DATA_BLOCK "Timer"   // DB2
{ S7_Optimized_Access := 'TRUE' }
VERSION : 0.0
// stored: AutoNumber false, IsOnlyStoredInLoadMemory false, IsRetainMemResEnabled false, IsWriteProtectedInAS false, MemoryReserve 100
   VAR
      T0 { S7_SetPoint := 'True'} : IEC_TIMER;   // Delay on pallet positioning
      T1 { S7_SetPoint := 'True'} : IEC_TIMER;   // Timer for acoustic siren
      T2 { S7_SetPoint := 'True'} : IEC_TIMER;   // Timer for restart after emergency
      T3 { S7_SetPoint := 'True'} : IEC_TIMER;   // Timer to reset emergency
      T4 { S7_SetPoint := 'True'} : IEC_TIMER;   // Timer to reset the cycles
      T5 { S7_SetPoint := 'True'} : IEC_TIMER;   // Delay for backward on table rotation inverter
      T6 { S7_SetPoint := 'True'} : IEC_TIMER;   // Delay for forward on table rotation inverter
      T7 { S7_SetPoint := 'True'} : IEC_TIMER;   // Timeout for table phase
      T8 { S7_SetPoint := 'True'} : IEC_TIMER;   // Table rotation speed timer
      T9 { S7_SetPoint := 'True'} : IEC_TIMER;   // Timer SA type for spool carriage motor
      T10 { S7_SetPoint := 'True'} : IEC_TIMER;   // Timer SA type for table rotation motor
      T11 { S7_SetPoint := 'True'} : IEC_TIMER;   // Timer SA type for spool carriage downward
      T12 { S7_SetPoint := 'True'} : IEC_TIMER;   // Timer SA type for spool carriage upward
      T13 { S7_SetPoint := 'True'} : IEC_TIMER;   // Timer SA type for top carriage motor
      T14 { S7_SetPoint := 'True'} : IEC_TIMER;   // Delay for forward on spool carriage and machine conveyor inverter
      T15 { S7_SetPoint := 'True'} : IEC_TIMER;   // Timer for lifter upward
      T16 { S7_SetPoint := 'True'} : IEC_TIMER;   // Timeout for pallet lifter upward/downward
      T17 { S7_SetPoint := 'True'} : IEC_TIMER;   // Time for pressure plate downward
      T18 { S7_SetPoint := 'True'} : IEC_TIMER;   // Timeout for pressure plate upward/downward
      T19 { S7_SetPoint := 'True'} : IEC_TIMER;   // Delay for backward on spool carriage and machine conveyor inverter
      T20 { S7_SetPoint := 'True'} : IEC_TIMER;   // Delay for table rotation deceleration
      T21 { S7_SetPoint := 'True'} : IEC_TIMER;   // Film broken delay for spool carriage
      T22 { S7_SetPoint := 'True'} : IEC_TIMER;   // Delay for pressure plate positioning on pallet
      T23 { S7_SetPoint := 'True'} : IEC_TIMER;   // Timer SA type for conveyor motor
      T24 { S7_SetPoint := 'True'} : IEC_TIMER;   // Delay on pallet positioning left
      T25 { S7_SetPoint := 'True'} : IEC_TIMER;   // Delay on machine conveyor stop
      T26 { S7_SetPoint := 'True'} : IEC_TIMER;   // Delay to load/unload pallet simultaneously
      T27 { S7_SetPoint := 'True'} : IEC_TIMER;   // Delay to have outfeed control free
      T28 { S7_SetPoint := 'True'} : IEC_TIMER;   // Timer for end of transfer signal
      T29 { S7_SetPoint := 'True'} : IEC_TIMER;   // Timer to check spool carriage encoder
      T30 { S7_SetPoint := 'True'} : IEC_TIMER;   // Timer to check spool carriage encoder
      T31 { S7_SetPoint := 'True'} : IEC_TIMER;   // Time to record spool carriage movement speed
      T32 { S7_SetPoint := 'True'} : IEC_TIMER;   // Timeout for single or lower(double) rope unit open/close
      T33 { S7_SetPoint := 'True'} : IEC_TIMER;   // Timer for outfeed rotating table control engaged
      T34 { S7_SetPoint := 'True'} : IEC_TIMER;   // Timer for prestretch restart
      T35 { S7_SetPoint := 'True'} : IEC_TIMER;   // Delay to open single or lower(double) rope unit
      T36 { S7_SetPoint := 'True'} : IEC_TIMER;   // Timeout for welder unit upward/downward
      T37 { S7_SetPoint := 'True'} : IEC_TIMER;   // Timeout for welder contrast downward
      T38 { S7_SetPoint := 'True'} : IEC_TIMER;   // Timeout for welder contrast upward
      T39 { S7_SetPoint := 'True'} : IEC_TIMER;   // Timeout for clamp upward/downward
      T40 { S7_SetPoint := 'True'} : IEC_TIMER;   // Timeout for clamp open/close
      T41 { S7_SetPoint := 'True'} : IEC_TIMER;   // Welding timer for welder
      T42 { S7_SetPoint := 'True'} : IEC_TIMER;   // Cutting timer
      T43 { S7_SetPoint := 'True'} : IEC_TIMER;   // Welder cooler timer
      T44 { S7_SetPoint := 'True'} : IEC_TIMER;   // Timer to check welder circuit 1 (current on)
      T45 { S7_SetPoint := 'True'} : IEC_TIMER;   // Timer to check welder circuit 2 (current off)
      T46 { S7_SetPoint := 'True'} : IEC_TIMER;   // Spring clamp up
      T47 { S7_SetPoint := 'True'} : IEC_TIMER;   // Welder contrast up
      T48 { S7_SetPoint := 'True'} : IEC_TIMER;   // Spring clamp open
      T49 { S7_SetPoint := 'True'} : IEC_TIMER;   // Welder and cut unit up
      T50 { S7_SetPoint := 'True'} : IEC_TIMER;   // Timer for encoder check
      T51 { S7_SetPoint := 'True'} : IEC_TIMER;   // Timer for display comunication control
      T52 { S7_SetPoint := 'True'} : IEC_TIMER;   // Timer to return to page 1 after 3 minutes
      T53 { S7_SetPoint := 'True'} : IEC_TIMER;   // Delay for test cycle
      T54 { S7_SetPoint := 'True'} : IEC_TIMER;   // Timer to reset infeed safety barrier
      T55 { S7_SetPoint := 'True'} : IEC_TIMER;   // Timer to reset infeed safety barrier
      T56 { S7_SetPoint := 'True'} : IEC_TIMER;   // Timer to reset outfeed safety barrier
      T57 { S7_SetPoint := 'True'} : IEC_TIMER;   // Timer to reset outfeed safety barrier
      T58 { S7_SetPoint := 'True'} : IEC_TIMER;   // Delay for infeed safety barrier muting photocell
      T59 { S7_SetPoint := 'True'} : IEC_TIMER;   // Delay for outfeed safety barrier muting photocell
      T60 { S7_SetPoint := 'True'} : IEC_TIMER;   // Delay for spool carriage downward for film tail
      T61 { S7_SetPoint := 'True'} : IEC_TIMER;   // Delay to open clamp during wrapping cycle
      T62 { S7_SetPoint := 'True'} : IEC_TIMER;   // Timer for table rotation forward on twist
      T63 { S7_SetPoint := 'True'} : IEC_TIMER;   // Timer SA type for top carriage upward
      T64 { S7_SetPoint := 'True'} : IEC_TIMER;   // Timer SA type for top carriage downward
      T65 { S7_SetPoint := 'True'} : IEC_TIMER;   // Delay on safety for top carriage movement
      T66 { S7_SetPoint := 'True'} : IEC_TIMER;   // Timer to check top film presence
      T67 { S7_SetPoint := 'True'} : IEC_TIMER;   // Timer to check top film presence
      T68 { S7_SetPoint := 'True'} : IEC_TIMER;   // Timeout for top film cutter forward/backward
      T69 { S7_SetPoint := 'True'} : IEC_TIMER;   // Timeout for clamp to lift top film open/close
      T70 { S7_SetPoint := 'True'} : IEC_TIMER;   // Timeout for clamp to block top film open/close
      T71 { S7_SetPoint := 'True'} : IEC_TIMER;   // Timeout for top carriage forward/backward movement
      T72 { S7_SetPoint := 'True'} : IEC_TIMER;   // Timeout for top carriage forward/backward movement
      T73 { S7_SetPoint := 'True'} : IEC_TIMER;   // Timeout for top carriage upward/downward movement
      T74 { S7_SetPoint := 'True'} : IEC_TIMER;   // Timeout for top carriage upward/downward movement
      T75 { S7_SetPoint := 'True'} : IEC_TIMER;   // Delay for spool carriage downward during top cycle
      T76 { S7_SetPoint := 'True'} : IEC_TIMER;   // Claw clamp closed
      T77 { S7_SetPoint := 'True'} : IEC_TIMER;   // Timeout for welder and cut unit forward/backward
      T78 { S7_SetPoint := 'True'} : IEC_TIMER;   // Delay to open upper(double) rope unit
      T79 { S7_SetPoint := 'True'} : IEC_TIMER;   // Timer SA type for table rotation brake
      T80 { S7_SetPoint := 'True'} : IEC_TIMER;   // Timer for spool carriage movement speed
      T81 { S7_SetPoint := 'True'} : IEC_TIMER;   // Claw clamp closed
      T82 { S7_SetPoint := 'True'} : IEC_TIMER;   // Timeout for welder and cut unit forward/backward
      T83 { S7_SetPoint := 'True'} : IEC_TIMER;   // Delay between airblow and clamp
      T84 { S7_SetPoint := 'True'} : IEC_TIMER;   // Timer for table rotation speed
      T85 { S7_SetPoint := 'True'} : IEC_TIMER;   // Delay on infeed conveyor stop
      T86 { S7_SetPoint := 'True'} : IEC_TIMER;   // Delay for prestretch during acceleration
      T87 { S7_SetPoint := 'True'} : IEC_TIMER;   // Timer for slow conveyor manual movement
      T88 { S7_SetPoint := 'True'} : IEC_TIMER;
      T89 { S7_SetPoint := 'True'} : IEC_TIMER;   // Timer for wrong pallet positioning without outfeed control
      T90 { S7_SetPoint := 'True'} : IEC_TIMER;   // Timer for spool carriage upward for table cycle
      T91 { S7_SetPoint := 'True'} : IEC_TIMER;   // Delay to close clamp after cutter forward
      T92 { S7_SetPoint := 'True'} : IEC_TIMER;   // Delay for contrast downward
      T93 { S7_SetPoint := 'True'} : IEC_TIMER;
      T94 { S7_SetPoint := 'True'} : IEC_TIMER;
      T95 { S7_SetPoint := 'True'} : IEC_TIMER;
      T96 { S7_SetPoint := 'True'} : IEC_TIMER;   // Timeout for fire door pos.4-5 opening
      T97 { S7_SetPoint := 'True'} : IEC_TIMER;   // Delay conveyor manual movement
      T98 { S7_SetPoint := 'True'} : IEC_TIMER;   // Delay start cycle pos.1
      T99 { S7_SetPoint := 'True'} : IEC_TIMER;   // Time to load with forklift
      T100 { S7_SetPoint := 'True'} : IEC_TIMER;   // Timer for end of pallet transfer in infeed signal
      T101 { S7_SetPoint := 'True'} : IEC_TIMER;   // Timeout for conveyor pos 01
      T102 { S7_SetPoint := 'True'} : IEC_TIMER;   // Time to load with forklift
      T103 { S7_SetPoint := 'True'} : IEC_TIMER;   // Timeout for conveyor pos 02
      T104 { S7_SetPoint := 'True'} : IEC_TIMER;
      T105 { S7_SetPoint := 'True'} : IEC_TIMER;   // Timeout for conveyor pos 04
      T106 { S7_SetPoint := 'True'} : IEC_TIMER;   // Timeout for conveyor pos 03
      T107 { S7_SetPoint := 'True'} : IEC_TIMER;   // Time for pallet unload with forklift
      T108 { S7_SetPoint := 'True'} : IEC_TIMER;   // Delay Button Stop cycle support memory
      T109 { S7_SetPoint := 'True'} : IEC_TIMER;   // Time for pallet load with forklift from reverse
      T110 { S7_SetPoint := 'True'} : IEC_TIMER;   // Timer to reset machine and cycle
      T111 { S7_SetPoint := 'True'} : IEC_TIMER;   // Delay timer for lifter pos.2 low position
      T112 { S7_SetPoint := 'True'} : IEC_TIMER;   // Delay timer for lifter pos.2 up position
      T113 { S7_SetPoint := 'True'} : IEC_TIMER;   // Delay timer pallet positioned on lifter pos.2
      T114 { S7_SetPoint := 'True'} : IEC_TIMER;   // Timer SA for lifter in top position
      T115 { S7_SetPoint := 'True'} : IEC_TIMER;   // Timeout for conveyor pos.2
      T116 { S7_SetPoint := 'True'} : IEC_TIMER;   // Timeout for lifter pos.2 upstroke
      T117 { S7_SetPoint := 'True'} : IEC_TIMER;   // Timeout for lifter pos.2 downstroke
      T118 { S7_SetPoint := 'True'} : IEC_TIMER;   // Timer to filter lifter pos.2 in up position
      T119 { S7_SetPoint := 'True'} : IEC_TIMER;
      T120 { S7_SetPoint := 'True'} : IEC_TIMER;   // Timer to check conveyor encoder
      T121 { S7_SetPoint := 'True'} : IEC_TIMER;   // Timer to check conveyor encoder
      T122 { S7_SetPoint := 'True'} : IEC_TIMER;
      T123 { S7_SetPoint := 'True'} : IEC_TIMER;
      T124 { S7_SetPoint := 'True'} : IEC_TIMER;
      T125 { S7_SetPoint := 'True'} : IEC_TIMER;
      T126 { S7_SetPoint := 'True'} : IEC_TIMER;
      T127 { S7_SetPoint := 'True'} : IEC_TIMER;   // Delay to have outfeed rotating arm control free from reverse
      T128 { S7_SetPoint := 'True'} : IEC_TIMER;   // Timer for end of transfer signal from reverse
      T129 { S7_SetPoint := 'True'} : IEC_TIMER;
      T130 { S7_SetPoint := 'True'} : IEC_TIMER;
      T131 { S7_SetPoint := 'True'} : IEC_TIMER;
      T132 { S7_SetPoint := 'True'} : IEC_TIMER;   // Timeout for single or lower(double) rope unit open/close
      T133 { S7_SetPoint := 'True'} : IEC_TIMER;
      T134 { S7_SetPoint := 'True'} : IEC_TIMER;
      T135 { S7_SetPoint := 'True'} : IEC_TIMER;   // Delay to open single or lower(double) rope unit
      T136 { S7_SetPoint := 'True'} : IEC_TIMER;
      T137 { S7_SetPoint := 'True'} : IEC_TIMER;
      T138 { S7_SetPoint := 'True'} : IEC_TIMER;
      T139 { S7_SetPoint := 'True'} : IEC_TIMER;   // Delay for top carriage forward stop (Top)
      T140 { S7_SetPoint := 'True'} : IEC_TIMER;   // Delay for top carriage backward stop (Top)
      T141 { S7_SetPoint := 'True'} : IEC_TIMER;
      T142 { S7_SetPoint := 'True'} : IEC_TIMER;   // Delay for top carriage down to release top film (Top)
      T143 { S7_SetPoint := 'True'} : IEC_TIMER;   // Delay to release top film from clamp (Top)
      T144 { S7_SetPoint := 'True'} : IEC_TIMER;   // Timer 1 for top film broken (Top)
      T145 { S7_SetPoint := 'True'} : IEC_TIMER;   // Timer 2 for top film broken (Top)
      T146 { S7_SetPoint := 'True'} : IEC_TIMER;   // Delay to stop top carriage forward for top film broken (Top)
      T147 { S7_SetPoint := 'True'} : IEC_TIMER;   // Delay to stop top carriage against vibration (Top)
      T148 { S7_SetPoint := 'True'} : IEC_TIMER;   // Timeout for top cutter (Top)
      T149 { S7_SetPoint := 'True'} : IEC_TIMER;   // Timeout for clamp to pull top film (Top)
      T150 { S7_SetPoint := 'True'} : IEC_TIMER;   // Timeout for clamp to block top film (Top)
      T151 { S7_SetPoint := 'True'} : IEC_TIMER;   // Timer SA type for top brake (Top)
      T152 { S7_SetPoint := 'True'} : IEC_TIMER;   // Timer for top brake control (Top)
      T153 { S7_SetPoint := 'True'} : IEC_TIMER;
      T154 { S7_SetPoint := 'True'} : IEC_TIMER;
      T155 { S7_SetPoint := 'True'} : IEC_TIMER;   // Timeout for conveyor pos 03
      T156 { S7_SetPoint := 'True'} : IEC_TIMER;   // Timeout for conveyor pos 04
      T157 { S7_SetPoint := 'True'} : IEC_TIMER;   // Timeout for conveyor pos 05
      T158 { S7_SetPoint := 'True'} : IEC_TIMER;   // Timeout for conveyor pos 06
      T159 { S7_SetPoint := 'True'} : IEC_TIMER;   // Timeout for conveyor pos 07
      T160 { S7_SetPoint := 'True'} : IEC_TIMER;   // Timeout for conveyor pos 08
      T161 { S7_SetPoint := 'True'} : IEC_TIMER;
      T162 { S7_SetPoint := 'True'} : IEC_TIMER;
      T163 { S7_SetPoint := 'True'} : IEC_TIMER;   // Watchdog timer for network communication
      T164 { S7_SetPoint := 'True'} : IEC_TIMER;
      T165 { S7_SetPoint := 'True'} : IEC_TIMER;
      T166 { S7_SetPoint := 'True'} : IEC_TIMER;
      T167 { S7_SetPoint := 'True'} : IEC_TIMER;
      T168 { S7_SetPoint := 'True'} : IEC_TIMER;
      T169 { S7_SetPoint := 'True'} : IEC_TIMER;
      T170 { S7_SetPoint := 'True'} : IEC_TIMER;
      T171 { S7_SetPoint := 'True'} : IEC_TIMER;
      T172 { S7_SetPoint := 'True'} : IEC_TIMER;
      T173 { S7_SetPoint := 'True'} : IEC_TIMER;
      T174 { S7_SetPoint := 'True'} : IEC_TIMER;
      T175 { S7_SetPoint := 'True'} : IEC_TIMER;
      T176 { S7_SetPoint := 'True'} : IEC_TIMER;
      T177 { S7_SetPoint := 'True'} : IEC_TIMER;
      T178 { S7_SetPoint := 'True'} : IEC_TIMER;
      T179 { S7_SetPoint := 'True'} : IEC_TIMER;   // Delay for top pallet height reading photocell (fast cycle)
      T180 { S7_SetPoint := 'True'} : IEC_TIMER;
      T181 { S7_SetPoint := 'True'} : IEC_TIMER;
      T182 { S7_SetPoint := 'True'} : IEC_TIMER;
      T183 { S7_SetPoint := 'True'} : IEC_TIMER;
      T184 { S7_SetPoint := 'True'} : IEC_TIMER;
      T185 { S7_SetPoint := 'True'} : IEC_TIMER;
      T186 { S7_SetPoint := 'True'} : IEC_TIMER;
      T187 { S7_SetPoint := 'True'} : IEC_TIMER;
      T188 { S7_SetPoint := 'True'} : IEC_TIMER;
      T189 { S7_SetPoint := 'True'} : IEC_TIMER;
      T190 { S7_SetPoint := 'True'} : IEC_TIMER;
      T191 { S7_SetPoint := 'True'} : IEC_TIMER;
      T192 { S7_SetPoint := 'True'} : IEC_TIMER;
      T193 { S7_SetPoint := 'True'} : IEC_TIMER;
      T194 { S7_SetPoint := 'True'} : IEC_TIMER;
      T195 { S7_SetPoint := 'True'} : IEC_TIMER;
      T196 { S7_SetPoint := 'True'} : IEC_TIMER;
      T197 { S7_SetPoint := 'True'} : IEC_TIMER;
      T198 { S7_SetPoint := 'True'} : IEC_TIMER;
      T199 { S7_SetPoint := 'True'} : IEC_TIMER;
      T200 { S7_SetPoint := 'True'} : IEC_TIMER;   // T_InverterAlarm - Time to filter inverter alarms
      T201 { S7_SetPoint := 'True'} : IEC_TIMER;   // T_ProfinetDiag - Time to filter 'DeviceStates' diagnostic output (Profinet)
      T202 { S7_SetPoint := 'True'} : IEC_TIMER;   // Timer for U201 start command (after enable)
      T203 { S7_SetPoint := 'True'} : IEC_TIMER;   // Timer table backward
      T204 { S7_SetPoint := 'True'} : IEC_TIMER;   // Timer ciclo fiera
      T205 { S7_SetPoint := 'True'} : IEC_TIMER;   // TON per OFF1 U201
      T206 { S7_SetPoint := 'True'} : IEC_TIMER;   // TOF per OFF1 U201
      T207 { S7_SetPoint := 'True'} : IEC_TIMER;   // Timer coppia tavola
      T208 { S7_SetPoint := 'True'} : IEC_TIMER;   // T_ModbusErrors
      T209 { S7_SetPoint := 'True'} : IEC_TIMER;
      T210 { S7_SetPoint := 'True'} : IEC_TIMER;   // Time to filter contrast back sensor
      T211 { S7_SetPoint := 'True'} : IEC_TIMER;   // Timeout for welder contrast forward
      T212 { S7_SetPoint := 'True'} : IEC_TIMER;   // Timeout for welder contrast backward
      T213 { S7_SetPoint := 'True'} : IEC_TIMER;   // Timeout for (double) full rope unit open/close
      T214 { S7_SetPoint := 'True'} : IEC_TIMER;   // Delay to open single or lower(double) rope unit
      T215 { S7_SetPoint := 'True'} : IEC_TIMER;   // Time Contrast Backward
      T216 { S7_SetPoint := 'True'} : IEC_TIMER;   // Time Contrast Manual forward
   END_VAR
BEGIN
   T0.PT := T#0MS;
   T0.IN := FALSE;
   T1.PT := T#1S_200MS;
   T1.IN := FALSE;
   T2.PT := T#6S;
   T2.IN := TRUE;
   T3.PT := T#700MS;
   T3.IN := FALSE;
   T4.PT := T#2S;
   T4.IN := FALSE;
   T5.PT := T#800MS;
   T5.IN := FALSE;
   T6.PT := T#800MS;
   T6.IN := FALSE;
   T7.PT := T#50S;
   T7.IN := FALSE;
   T8.PT := T#1M_39S;
   T8.IN := FALSE;
   T9.PT := T#700MS;
   T9.IN := FALSE;
   T10.PT := T#2S;
   T10.IN := FALSE;
   T11.PT := T#500MS;
   T11.IN := FALSE;
   T12.PT := T#500MS;
   T12.IN := FALSE;
   T13.PT := T#0MS;
   T13.IN := FALSE;
   T14.PT := T#200MS;
   T14.IN := FALSE;
   T15.PT := T#0MS;
   T15.IN := FALSE;
   T16.PT := T#0MS;
   T16.IN := FALSE;
   T17.PT := T#0MS;
   T17.IN := FALSE;
   T18.PT := T#0MS;
   T18.IN := FALSE;
   T19.PT := T#200MS;
   T19.IN := FALSE;
   T20.PT := T#0MS;
   T20.IN := FALSE;
   T21.PT := T#2S;
   T21.IN := FALSE;
   T22.PT := T#0MS;
   T22.IN := FALSE;
   T23.PT := T#0MS;
   T23.IN := FALSE;
   T24.PT := T#0MS;
   T24.IN := FALSE;
   T25.PT := T#0MS;
   T25.IN := FALSE;
   T26.PT := T#0MS;
   T26.IN := FALSE;
   T27.PT := T#1S_500MS;
   T27.IN := TRUE;
   T28.PT := T#2S;
   T28.IN := TRUE;
   T29.PT := T#0MS;
   T29.IN := FALSE;
   T30.PT := T#3S;
   T30.IN := FALSE;
   T31.PT := T#0MS;
   T31.IN := FALSE;
   T32.PT := T#0MS;
   T32.IN := FALSE;
   T33.PT := T#0MS;
   T33.IN := FALSE;
   T34.PT := T#0MS;
   T34.IN := FALSE;
   T35.PT := T#0MS;
   T35.IN := FALSE;
   T36.PT := T#0MS;
   T36.IN := FALSE;
   T37.PT := T#0MS;
   T37.IN := FALSE;
   T38.PT := T#10S;
   T38.IN := FALSE;
   T39.PT := T#0MS;
   T39.IN := FALSE;
   T40.PT := T#0MS;
   T40.IN := FALSE;
   T41.PT := T#650MS;
   T41.IN := FALSE;
   T42.PT := T#3S;
   T42.IN := FALSE;
   T43.PT := T#0MS;
   T43.IN := FALSE;
   T44.PT := T#3S_500MS;
   T44.IN := FALSE;
   T45.PT := T#1S;
   T45.IN := FALSE;
   T46.PT := T#0MS;
   T46.IN := FALSE;
   T47.PT := T#500MS;
   T47.IN := TRUE;
   T48.PT := T#0MS;
   T48.IN := FALSE;
   T49.PT := T#0MS;
   T49.IN := FALSE;
   T50.PT := T#0MS;
   T50.IN := FALSE;
   T51.PT := T#4S;
   T51.IN := TRUE;
   T52.PT := T#0MS;
   T52.IN := FALSE;
   T53.PT := T#0MS;
   T53.IN := TRUE;
   T54.PT := T#0MS;
   T54.IN := FALSE;
   T55.PT := T#0MS;
   T55.IN := FALSE;
   T56.PT := T#0MS;
   T56.IN := FALSE;
   T57.PT := T#0MS;
   T57.IN := FALSE;
   T58.PT := T#0MS;
   T58.IN := FALSE;
   T59.PT := T#0MS;
   T59.IN := FALSE;
   T60.PT := T#0MS;
   T60.IN := FALSE;
   T61.PT := T#0MS;
   T61.IN := FALSE;
   T62.PT := T#0MS;
   T62.IN := FALSE;
   T63.PT := T#0MS;
   T63.IN := FALSE;
   T64.PT := T#0MS;
   T64.IN := FALSE;
   T65.PT := T#0MS;
   T65.IN := FALSE;
   T66.PT := T#0MS;
   T66.IN := FALSE;
   T67.PT := T#0MS;
   T67.IN := FALSE;
   T68.PT := T#0MS;
   T68.IN := FALSE;
   T69.PT := T#0MS;
   T69.IN := FALSE;
   T70.PT := T#0MS;
   T70.IN := FALSE;
   T71.PT := T#0MS;
   T71.IN := FALSE;
   T72.PT := T#0MS;
   T72.IN := FALSE;
   T73.PT := T#0MS;
   T73.IN := FALSE;
   T74.PT := T#0MS;
   T74.IN := FALSE;
   T75.PT := T#0MS;
   T75.IN := FALSE;
   T76.PT := T#0MS;
   T76.IN := FALSE;
   T77.PT := T#0MS;
   T77.IN := FALSE;
   T78.PT := T#0MS;
   T78.IN := FALSE;
   T79.PT := T#2S;
   T79.IN := FALSE;
   T80.PT := T#1S;
   T80.IN := TRUE;
   T81.PT := T#700MS;
   T81.IN := TRUE;
   T82.PT := T#10S;
   T82.IN := FALSE;
   T83.PT := T#500MS;
   T83.IN := FALSE;
   T84.PT := T#400MS;
   T84.IN := TRUE;
   T85.PT := T#0MS;
   T85.IN := FALSE;
   T86.PT := T#300MS;
   T86.IN := FALSE;
   T87.PT := T#0MS;
   T87.IN := FALSE;
   T88.PT := T#0MS;
   T88.IN := FALSE;
   T89.PT := T#0MS;
   T89.IN := FALSE;
   T90.PT := T#2S;
   T90.IN := FALSE;
   T91.PT := T#1S;
   T91.IN := FALSE;
   T92.PT := T#0MS;
   T92.IN := FALSE;
   T93.PT := T#0MS;
   T93.IN := FALSE;
   T94.PT := T#0MS;
   T94.IN := FALSE;
   T95.PT := T#0MS;
   T95.IN := FALSE;
   T96.PT := T#0MS;
   T96.IN := FALSE;
   T97.PT := T#0MS;
   T97.IN := FALSE;
   T98.PT := T#0MS;
   T98.IN := FALSE;
   T99.PT := T#0MS;
   T99.IN := FALSE;
   T100.PT := T#0MS;
   T100.IN := FALSE;
   T101.PT := T#0MS;
   T101.IN := FALSE;
   T102.PT := T#0MS;
   T102.IN := FALSE;
   T103.PT := T#0MS;
   T103.IN := FALSE;
   T104.PT := T#0MS;
   T104.IN := FALSE;
   T105.PT := T#0MS;
   T105.IN := FALSE;
   T106.PT := T#0MS;
   T106.IN := FALSE;
   T107.PT := T#0MS;
   T107.IN := FALSE;
   T108.PT := T#0MS;
   T108.IN := FALSE;
   T109.PT := T#0MS;
   T109.IN := FALSE;
   T110.PT := T#0MS;
   T110.IN := FALSE;
   T111.PT := T#0MS;
   T111.IN := FALSE;
   T112.PT := T#0MS;
   T112.IN := FALSE;
   T113.PT := T#0MS;
   T113.IN := FALSE;
   T114.PT := T#0MS;
   T114.IN := FALSE;
   T115.PT := T#0MS;
   T115.IN := FALSE;
   T116.PT := T#0MS;
   T116.IN := FALSE;
   T117.PT := T#0MS;
   T117.IN := FALSE;
   T118.PT := T#0MS;
   T118.IN := FALSE;
   T119.PT := T#0MS;
   T119.IN := FALSE;
   T120.PT := T#0MS;
   T120.IN := FALSE;
   T121.PT := T#0MS;
   T121.IN := FALSE;
   T122.PT := T#0MS;
   T122.IN := FALSE;
   T123.PT := T#0MS;
   T123.IN := FALSE;
   T124.PT := T#0MS;
   T124.IN := FALSE;
   T125.PT := T#0MS;
   T125.IN := FALSE;
   T126.PT := T#0MS;
   T126.IN := FALSE;
   T127.PT := T#0MS;
   T127.IN := FALSE;
   T128.PT := T#0MS;
   T128.IN := FALSE;
   T129.PT := T#0MS;
   T129.IN := FALSE;
   T130.PT := T#0MS;
   T130.IN := FALSE;
   T131.PT := T#0MS;
   T131.IN := FALSE;
   T132.PT := T#3S;
   T132.IN := FALSE;
   T133.PT := T#0MS;
   T133.IN := FALSE;
   T134.PT := T#0MS;
   T134.IN := FALSE;
   T135.PT := T#1S_500MS;
   T135.IN := TRUE;
   T136.PT := T#0MS;
   T136.IN := FALSE;
   T137.PT := T#0MS;
   T137.IN := FALSE;
   T138.PT := T#0MS;
   T138.IN := FALSE;
   T139.PT := T#0MS;
   T139.IN := FALSE;
   T140.PT := T#0MS;
   T140.IN := FALSE;
   T141.PT := T#0MS;
   T141.IN := FALSE;
   T142.PT := T#0MS;
   T142.IN := FALSE;
   T143.PT := T#0MS;
   T143.IN := FALSE;
   T144.PT := T#0MS;
   T144.IN := FALSE;
   T145.PT := T#0MS;
   T145.IN := FALSE;
   T146.PT := T#0MS;
   T146.IN := FALSE;
   T147.PT := T#0MS;
   T147.IN := FALSE;
   T148.PT := T#0MS;
   T148.IN := FALSE;
   T149.PT := T#0MS;
   T149.IN := FALSE;
   T150.PT := T#0MS;
   T150.IN := FALSE;
   T151.PT := T#0MS;
   T151.IN := FALSE;
   T152.PT := T#0MS;
   T152.IN := FALSE;
   T153.PT := T#0MS;
   T153.IN := FALSE;
   T154.PT := T#0MS;
   T154.IN := FALSE;
   T155.PT := T#0MS;
   T155.IN := FALSE;
   T156.PT := T#0MS;
   T156.IN := FALSE;
   T157.PT := T#0MS;
   T157.IN := FALSE;
   T158.PT := T#0MS;
   T158.IN := FALSE;
   T159.PT := T#0MS;
   T159.IN := FALSE;
   T160.PT := T#0MS;
   T160.IN := FALSE;
   T161.PT := T#0MS;
   T161.IN := FALSE;
   T162.PT := T#0MS;
   T162.IN := FALSE;
   T163.PT := T#0MS;
   T163.IN := FALSE;
   T164.PT := T#0MS;
   T164.IN := FALSE;
   T165.PT := T#0MS;
   T165.IN := FALSE;
   T166.PT := T#0MS;
   T166.IN := FALSE;
   T167.PT := T#0MS;
   T167.IN := FALSE;
   T168.PT := T#0MS;
   T168.IN := FALSE;
   T169.PT := T#0MS;
   T169.IN := FALSE;
   T170.PT := T#0MS;
   T170.IN := FALSE;
   T171.PT := T#0MS;
   T171.IN := FALSE;
   T172.PT := T#0MS;
   T172.IN := FALSE;
   T173.PT := T#0MS;
   T173.IN := FALSE;
   T174.PT := T#0MS;
   T174.IN := FALSE;
   T175.PT := T#0MS;
   T175.IN := FALSE;
   T176.PT := T#0MS;
   T176.IN := FALSE;
   T177.PT := T#0MS;
   T177.IN := FALSE;
   T178.PT := T#0MS;
   T178.IN := FALSE;
   T179.PT := T#0MS;
   T179.IN := FALSE;
   T180.PT := T#0MS;
   T180.IN := FALSE;
   T181.PT := T#0MS;
   T181.IN := FALSE;
   T182.PT := T#0MS;
   T182.IN := FALSE;
   T183.PT := T#0MS;
   T183.IN := FALSE;
   T184.PT := T#0MS;
   T184.IN := FALSE;
   T185.PT := T#0MS;
   T185.IN := FALSE;
   T186.PT := T#0MS;
   T186.IN := FALSE;
   T187.PT := T#0MS;
   T187.IN := FALSE;
   T188.PT := T#0MS;
   T188.IN := FALSE;
   T189.PT := T#0MS;
   T189.IN := FALSE;
   T190.PT := T#0MS;
   T190.IN := FALSE;
   T191.PT := T#0MS;
   T191.IN := FALSE;
   T192.PT := T#0MS;
   T192.IN := FALSE;
   T193.PT := T#0MS;
   T193.IN := FALSE;
   T194.PT := T#0MS;
   T194.IN := FALSE;
   T195.PT := T#0MS;
   T195.IN := FALSE;
   T196.PT := T#0MS;
   T196.IN := FALSE;
   T197.PT := T#0MS;
   T197.IN := FALSE;
   T198.PT := T#0MS;
   T198.IN := FALSE;
   T199.PT := T#0MS;
   T199.IN := FALSE;
   T200.PT := T#5S;
   T200.IN := FALSE;
   T201.PT := T#200MS;
   T201.IN := TRUE;
   T202.PT := T#200MS;
   T202.IN := FALSE;
   T203.PT := T#1S;
   T203.IN := FALSE;
   T204.PT := T#0MS;
   T204.IN := FALSE;
   T205.PT := T#200MS;
   T205.IN := FALSE;
   T206.PT := T#200MS;
   T206.IN := FALSE;
   T207.PT := T#200MS;
   T207.IN := TRUE;
   T208.PT := T#0MS;
   T208.IN := FALSE;
   T209.PT := T#0MS;
   T209.IN := FALSE;
   T210.PT := T#200MS;
   T210.IN := FALSE;
   T211.PT := T#10S;
   T211.IN := FALSE;
   T212.PT := T#0MS;
   T212.IN := FALSE;
   T213.PT := T#3S;
   T213.IN := FALSE;
   T214.PT := T#1S_500MS;
   T214.IN := TRUE;
   T215.PT := T#2S;
   T215.IN := FALSE;
   T216.PT := T#5S;
   T216.IN := FALSE;
END_DATA_BLOCK

DATA_BLOCK "Alarmes"   // DB13
{ S7_Optimized_Access := 'TRUE' }
VERSION : 0.1
// stored: AutoNumber true, IsOnlyStoredInLoadMemory false, IsRetainMemResEnabled false, IsWriteProtectedInAS false, MemoryReserve 100
   VAR
      ALARMES_1 : Word;
      ALARMES_2 : Word;
      ALARME_DISPARO : Bool;
      PRESSÃO_MÁX : Bool;
      XV102_NÃO_ABRIU : Bool;
      XV102_NÃO_FECHOU : Bool;
   END_VAR
   VAR RETAIN
      TEMP_ABERT_XV102 : Time;
      TEMP_FECHO_XV102 : Time;
   END_VAR
BEGIN
END_DATA_BLOCK

DATA_BLOCK "Info_Ciclo"   // DB10
{ S7_Optimized_Access := 'TRUE' }
VERSION : 0.1
// stored: AutoNumber true, IsOnlyStoredInLoadMemory false, IsRetainMemResEnabled false, IsWriteProtectedInAS false, MemoryReserve 100
   VAR RETAIN
      LS101_SR : Bool;
   END_VAR
   VAR
      ESTADO_CICLO : Bool;
      CONTAGEM_CICLOS : Int;
      LIMITE_CONTAGEM : Bool;
   END_VAR
BEGIN
END_DATA_BLOCK

DATA_BLOCK "Analógicas"   // DB12
{ S7_Optimized_Access := 'TRUE' }
VERSION : 0.1
// stored: AutoNumber true, IsOnlyStoredInLoadMemory false, IsRetainMemResEnabled false, IsWriteProtectedInAS false, MemoryReserve 100
   VAR
      CAUDAL_FQ301 : Real;
      PRESSÃO_PC401 : Real;
   END_VAR
BEGIN
END_DATA_BLOCK

DATA_BLOCK "Estados_HMI_DB"   // DB15
{ S7_Optimized_Access := 'TRUE' }
VERSION : 0.1
// stored: AutoNumber true, IsOnlyStoredInLoadMemory false, IsRetainMemResEnabled false, IsWriteProtectedInAS false, MemoryReserve 100
   VAR
      MX201 : Bool;
      MX601 : Bool;
      XV101 : Bool;
      XV102 : Bool;
      BD601 : Bool;
      BD602 : Bool;
      BH201 : Bool;
      PH201 : Bool;
      RH201 : Bool;
      MX603 : Bool;
      BD603 : Bool;
      MX301 : Bool;
      PH301 : Bool;
      BM401 : Bool;
      MX604 : Bool;
      BD604 : Bool;
      MX605 : Bool;
      BD605 : Bool;
      BS001A : Bool;
      BS001B : Bool;
      BS501 : Bool;
      T_ATUAL_AREJAMENTO : Time;
      T_ATUAL_REDUÇÃO : Time;
      T_ATUAL_PRECIPITAÇÃO : Time;
      T_ATUAL_ALARME_PC401 : Time;
      T_ATUAL_COAG : Time;
      T_ATUAL_HISTERESE : Time;
   END_VAR
BEGIN
END_DATA_BLOCK

DATA_BLOCK "Inputs_HMI"   // DB14
{ S7_Optimized_Access := 'TRUE' }
VERSION : 0.1
// stored: AutoNumber true, IsOnlyStoredInLoadMemory false, IsRetainMemResEnabled false, IsWriteProtectedInAS false, MemoryReserve 100
   VAR RETAIN
      MODO_1 : Bool;
      MODO_2 : Bool;
   END_VAR
   VAR
      RESET_ALARME : Bool;
      START_CICLO : Bool;
   END_VAR
   VAR RETAIN
      MAN_AUTO : Bool;
   END_VAR
   VAR
      ON_OFF_MX201 : Bool;
      ON_OFF_MX301 : Bool;
      ON_OFF_MX601 : Bool;
      ON_OFF_MX603 : Bool;
      ON_OFF_MX604 : Bool;
      ON_OFF_MX605 : Bool;
      ON_OFF_BD601 : Bool;
      ON_OFF_BD602 : Bool;
      ON_OFF_BD603 : Bool;
      ON_OFF_BD604 : Bool;
      ON_OFF_BD605 : Bool;
      ON_OFF_BS001A : Bool;
      ON_OFF_BS001B : Bool;
      ON_OFF_BS501 : Bool;
      ON_OFF_BH201 : Bool;
      ON_OFF_BM401 : Bool;
      ON_OFF_XV101 : Bool;
      ON_OFF_XV102 : Bool;
   END_VAR
   VAR RETAIN
      TEMP_AREJAMENTO : Time := T#0m;
      TEMP_REDUÇÃO : Time := T#0m;
      TEMP_PRECIPITAÇÃO : Time := T#0m;
      TEMP_ALARME : Time := T#0m;
      TEMP_DOS_COAG : Time;
      HISTERESE : Time;
      SETPOINT_PC401 : Real;
      SP_LSH_TK02 : Real;
      SP_LSM_TK02 : Real;
      SP_LSL_TK02 : Real;
      SP_LSH_TK03 : Real;
      SP_LSM_TK03 : Real;
      SP_LSL_TK03 : Real;
   END_VAR
   VAR
      SALTAR_HISTERESE : Bool;
      RESET_CONT_CICLOS : Bool;
   END_VAR
   VAR RETAIN
      ENABLE_DISABLE_BD603 : Bool := true;
      SUSPENSÃO_CICLO_PRENSA : Bool;
      IGNORAR_LSH101_LSH501 : Bool;
   END_VAR
BEGIN
END_DATA_BLOCK

DATA_BLOCK "Níveis_TK02_TK03"   // DB11
{ S7_Optimized_Access := 'TRUE' }
VERSION : 0.1
// stored: AutoNumber true, IsOnlyStoredInLoadMemory false, IsRetainMemResEnabled false, IsWriteProtectedInAS false, MemoryReserve 100
   VAR
      LSH301 : Bool;
      LSM301 : Bool;
   END_VAR
   VAR RETAIN
      LSL301 : Bool;
   END_VAR
   VAR
      LSH201 : Bool;
      LSM201 : Bool;
      LSL201 : Bool;
      NÍVEL_EM_METROS_TK03 : Real;
      NÍVEL_EM_METROS_TK02 : Real;
   END_VAR
BEGIN
END_DATA_BLOCK

DATA_BLOCK "Etapas_Grafcet_1"   // DB4
{ S7_Optimized_Access := 'TRUE' }
VERSION : 0.1
// stored: AutoNumber true, IsOnlyStoredInLoadMemory false, IsRetainMemResEnabled false, IsWriteProtectedInAS false, MemoryReserve 100
   VAR RETAIN
      ETAPA_1 : Bool;
      ETAPA_2 : Bool;
      ETAPA_3 : Bool;
      ETAPA_4 : Bool;
      ETAPA_5 : Bool;
      ETAPA_6 : Bool;
      ETAPA_7 : Bool;
      ETAPA_8 : Bool;
      ETAPA_9 : Bool;
      ETAPA_33 : Bool;
      ETAPA_55 : Bool;
      RESET_ETAPA_1 : Bool;
      SUSPENSÃO_CICLO : Bool;
   END_VAR
BEGIN
END_DATA_BLOCK

DATA_BLOCK "Etapas_Grafcet_2"   // DB1
{ S7_Optimized_Access := 'TRUE' }
VERSION : 0.1
// stored: AutoNumber true, IsOnlyStoredInLoadMemory false, IsRetainMemResEnabled false, IsWriteProtectedInAS false, MemoryReserve 100
   VAR RETAIN
      ETAPA_10 : Bool;
      ETAPA_11 : Bool;
      ETAPA_12 : Bool;
      RESET_ETAPA_10 : Bool;
   END_VAR
BEGIN
END_DATA_BLOCK

DATA_BLOCK "Etapas_Grafcet_3"   // DB3
{ S7_Optimized_Access := 'TRUE' }
VERSION : 0.1
// stored: AutoNumber true, IsOnlyStoredInLoadMemory false, IsRetainMemResEnabled false, IsWriteProtectedInAS false, MemoryReserve 100
   VAR RETAIN
      ETAPA_13 : Bool;
      ETAPA_14 : Bool;
      ETAPA_15 : Bool;
      RESET_ETAPA_13 : Bool;
   END_VAR
BEGIN
END_DATA_BLOCK

DATA_BLOCK "Dados_Bombas"   // DB11
{ S7_Optimized_Access := 'TRUE' }
VERSION : 0.1
// stored: AutoNumber true, IsOnlyStoredInLoadMemory false, IsRetainMemResEnabled false, IsWriteProtectedInAS false, MemoryReserve 100
   VAR
      CONV_T_ALTERNANCIA_BOMBAS : Time;
      HORAS_TON_B2 : Int;
      HORAS_TON_B3 : Int;
      HORAS_TON_B1 : Int;
   END_VAR
BEGIN
END_DATA_BLOCK

DATA_BLOCK "Estados_HMI"   // DB18
{ S7_Optimized_Access := 'TRUE' }
VERSION : 0.1
// stored: AutoNumber true, IsOnlyStoredInLoadMemory false, IsRetainMemResEnabled false, IsWriteProtectedInAS false, MemoryReserve 100
   VAR
      "EV1.1_ESTADO" : Int;
      "EV2.1_ESTADO" : Int;
      "EV3.1_ESTADO" : Int;
      "EV4.1_ESTADO" : Int;
      "EV5.1_ESTADO" : Int;
      "EV1.2_ESTADO" : Int;
      "EV2.2_ESTADO" : Int;
      "EV3.2_ESTADO" : Int;
      "EV4.2_ESTADO" : Int;
      "EV5.2_ESTADO" : Int;
      "EV1.1_ESTADO_PAGCMD" : Int;
      "EV2.1_ESTADO_PAGCMD" : Int;
      "EV3.1_ESTADO_PAGCMD" : Int;
      "EV4.1_ESTADO_PAGCMD" : Int;
      "EV5.1_ESTADO_PAGCMD" : Int;
      "EV1.2_ESTADO_PAGCMD" : Int;
      "EV2.2_ESTADO_PAGCMD" : Int;
      "EV3.2_ESTADO_PAGCMD" : Int;
      "EV4.2_ESTADO_PAGCMD" : Int;
      "EV5.2_ESTADO_PAGCMD" : Int;
      BOMBA_1_ESTADO : Int;
      BOMBA_2_ESTADO : Int;
      BOMBA_3_ESTADO : Int;
      BOMBA_1_ESTADO_PAGCMD : Int;
      BOMBA_2_ESTADO_PAGCMD : Int;
      BOMBA_3_ESTADO_PAGCMD : Int;
      T_LAV_MINUTOS : Int;
      T_RINSE_MINUTOS : Int;
      ALARMES_LISTA_1 : Word;
      ALARMES_LISTA_2 : Word;
      ALARMES_LISTA_3 : Word;
   END_VAR
BEGIN
END_DATA_BLOCK

DATA_BLOCK "Dados_Ciclo"   // DB7
{ S7_Optimized_Access := 'TRUE' }
VERSION : 0.1
// stored: AutoNumber true, IsOnlyStoredInLoadMemory false, IsRetainMemResEnabled false, IsWriteProtectedInAS false, MemoryReserve 100
   VAR
      HOLD_ETAPA_1 : Bool;
   END_VAR
   VAR RETAIN
      FILTRO1_EM_CICLO : Bool;
      FILTRO2_EM_CICLO : Bool;
      FECHO_FILT_1 : Bool;
      FECHO_FILT_2 : Bool;
      ETAPA_ANTERIOR : Int := 1;
   END_VAR
   VAR
      ETAPA_N : Bool;
      POS_EVS_FILT_1 : String;
      POS_EVS_FILT_2 : String;
      PRESS_SP_FILT_1 : Bool;
      PRESS_SP_FILT_2 : Bool;
   END_VAR
   VAR RETAIN
      STOP_CICLO : Bool;
   END_VAR
   VAR
      AGEND_FILT_1 : Bool;
      AGEND_FILT_2 : Bool;
   END_VAR
   VAR RETAIN
      HORA_INIC_FILT_1 : USInt;
      MIN_INIC_FILT_1 : USInt;
      HORA_INIC_FILT_2 : USInt;
      MIN_INIC_FILT_2 : USInt;
      ENABLE_AGEND_FILT_1 : Bool;
      ENABLE_AGEND_FILT_2 : Bool;
   END_VAR
   VAR
      PRESSÃO_FILT1 : Real;
      PRESSÃO_FILT2 : Real;
   END_VAR
BEGIN
END_DATA_BLOCK

DATA_BLOCK "Etapas_Grafcet"   // DB1
{ S7_Optimized_Access := 'TRUE' }
VERSION : 0.1
// stored: AutoNumber true, IsOnlyStoredInLoadMemory false, IsRetainMemResEnabled false, IsWriteProtectedInAS false, MemoryReserve 100
   VAR
      ETAPA_1 : Bool;
      ETAPA_2 : Bool;
      ETAPA_3 : Bool;
      ETAPA_4 : Bool;
      ETAPA_5 : Bool;
      ETAPA_6 : Bool;
      ETAPA_7 : Bool;
      ETAPA_8 : Bool;
      ETAPA_9 : Bool;
      ETAPA_10 : Bool;
      ETAPA_11 : Bool;
      ETAPA_12 : Bool;
      ETAPA_13 : Bool;
      ETAPA_14 : Bool;
      ETAPA_15 : Bool := true;
      ETAPA_16 : Bool;
   END_VAR
BEGIN
END_DATA_BLOCK

DATA_BLOCK "System_Time"   // DB40
{ S7_Optimized_Access := 'TRUE' }
VERSION : 0.1
// stored: AutoNumber true, IsOnlyStoredInLoadMemory false, IsRetainMemResEnabled false, IsWriteProtectedInAS false, MemoryReserve 100
   VAR
      REAL_TIME_DATA : DTL;
   END_VAR
BEGIN
END_DATA_BLOCK

ORGANIZATION_BLOCK "Main"   // OB1, LAD, ProgramCycle
TITLE = "Main Program Sweep (Cycle)"
{ S7_Optimized_Access := 'TRUE' }
VERSION : 0.1
// stored: AutoNumber true, IsIECCheckEnabled false, SetENOAutomatically false
   VAR_INPUT
      Initial_Call : Bool;   // Initial call of this OB
      Remanence : Bool;   // =True, if remanent data are available
   END_VAR
BEGIN
END_ORGANIZATION_BLOCK

ORGANIZATION_BLOCK "Startup"   // OB100, LAD, Startup
TITLE = "Complete Restart"
{ S7_Optimized_Access := 'TRUE' }
VERSION : 0.1
// stored: AutoNumber false, IsIECCheckEnabled false, SetENOAutomatically false
   VAR_INPUT
      LostRetentive : Bool;   // True if retentive data are lost
      LostRTC : Bool;   // True if date and time are lost
   END_VAR
BEGIN

REGION Network 1: First cycle
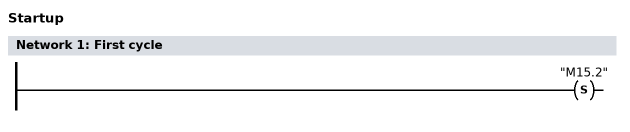
   RUNG wire#powerrail
      S_Coil( "M15.2" )
   END_RUNG
   // the same network as SCL:
   "M15.2" := TRUE;
END_REGION
END_ORGANIZATION_BLOCK

ORGANIZATION_BLOCK "Cyclic interrupt"   // OB30, LAD, CyclicInterrupt
TITLE = Rampa tiro
{ S7_Optimized_Access := 'TRUE' }
VERSION : 0.1
// Rampa per raggiungere tiro obiettivo e zero (0-20@100ms;20-100@20ms->3600ms)
// stored: AutoNumber true, IsIECCheckEnabled false, SetENOAutomatically false
   VAR_INPUT
      Initial_Call : Bool;   // Initial call of this OB
      Event_Count : Int;   // Events discarded
   END_VAR
   VAR_TEMP
      TempDint : DInt;
      TempDint_2 : DInt;
      TempInt : Int;
   END_VAR
   VAR_TEMP   // added for the SCL form of the ladder/FBD networks
      _w1 : Bool;
      _w2 : Bool;
   END_VAR
BEGIN

REGION Network 1: Impulso ogni 20ms (OB30)
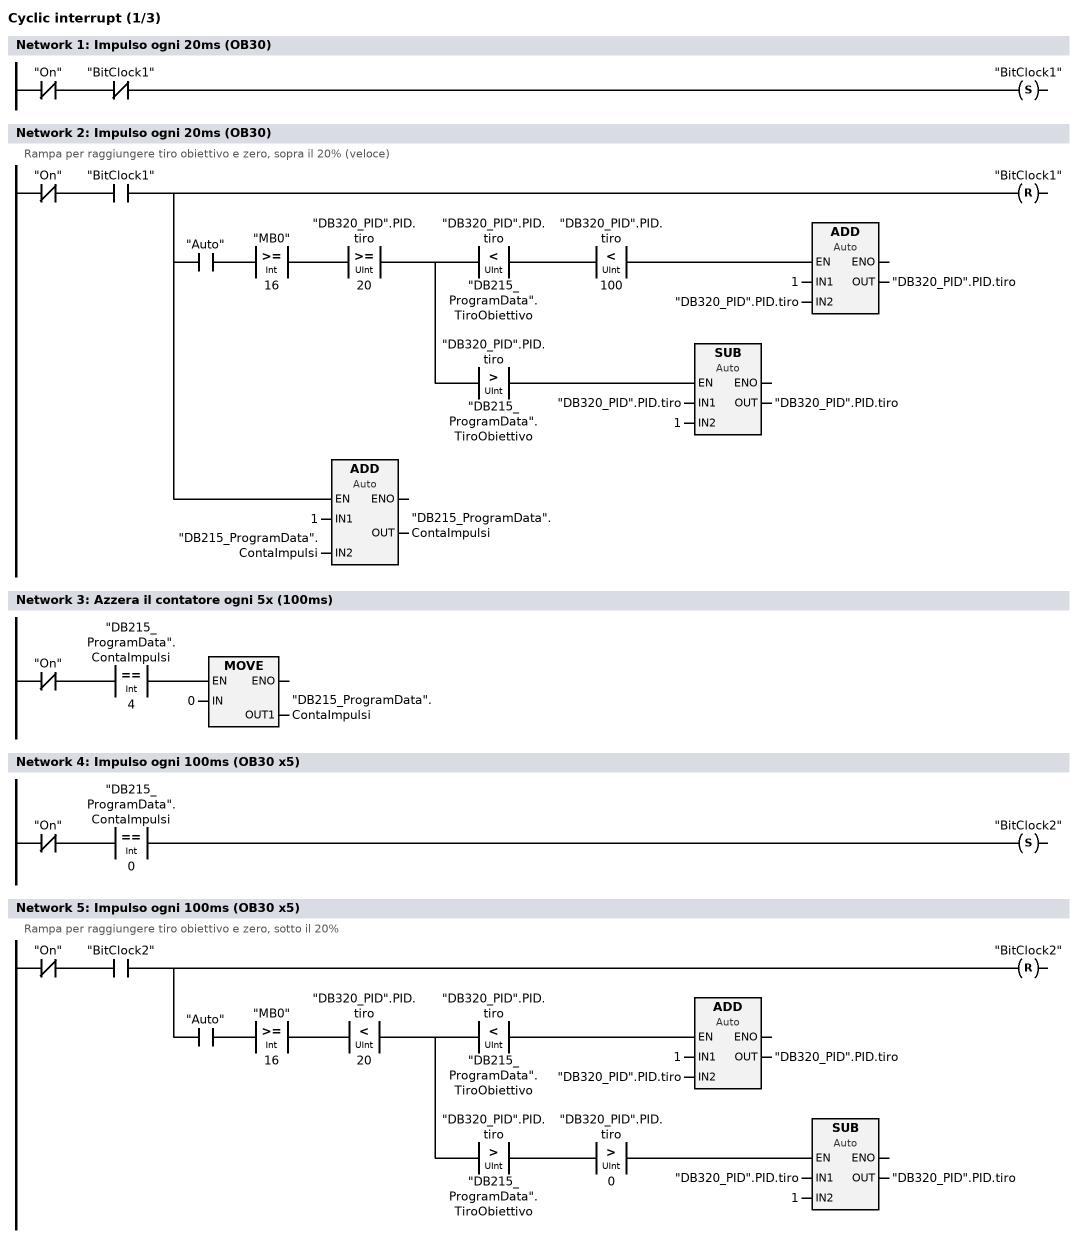
   RUNG wire#powerrail
      I_Contact( "On" )
      I_Contact( "BitClock1" )
      S_Coil( "BitClock1" )
   END_RUNG
   // the same network as SCL:
   IF NOT "On" AND NOT "BitClock1" THEN "BitClock1" := TRUE; END_IF;
END_REGION

REGION Network 2: Impulso ogni 20ms (OB30)
   // Rampa per raggiungere tiro obiettivo e zero, sopra il 20% (veloce)
   RUNG wire#powerrail
      I_Contact( "On" )
      Contact( "BitClock1" )
      wire#w1
      R_Coil( "BitClock1" )
   END_RUNG
   RUNG wire#w1
      Contact( "Auto" )
      { S7_Templates := "SrcType := Int" } GE_Contact(in1 := "MB0", in2 := 16)
      { S7_Templates := "SrcType := UInt" } GE_Contact(in1 := "DB320_PID".PID.tiro, in2 := 20)
      wire#w2
      { S7_Templates := "SrcType := UInt" } LT_Contact(in1 := "DB320_PID".PID.tiro, in2 := "DB215_ProgramData".TiroObiettivo)
      { S7_Templates := "SrcType := UInt" } LT_Contact(in1 := "DB320_PID".PID.tiro, in2 := 100)
      Add(in1 := 1, in2 := "DB320_PID".PID.tiro, out => "DB320_PID".PID.tiro)
   END_RUNG
   RUNG wire#w2
      { S7_Templates := "SrcType := UInt" } GT_Contact(in1 := "DB320_PID".PID.tiro, in2 := "DB215_ProgramData".TiroObiettivo)
      Sub(in1 := "DB320_PID".PID.tiro, in2 := 1, out => "DB320_PID".PID.tiro)
   END_RUNG
   RUNG wire#w1
      Add(in1 := 1, in2 := "DB215_ProgramData".ContaImpulsi, out => "DB215_ProgramData".ContaImpulsi)
   END_RUNG
   // the same network as SCL:
   #_w1 := NOT "On" AND "BitClock1";
   IF #_w1 THEN "BitClock1" := FALSE; END_IF;
   #_w2 := #_w1 AND "Auto" AND ("MB0" >= 16) AND ("DB320_PID".PID.tiro >= 20);
   IF #_w2 AND ("DB320_PID".PID.tiro < "DB215_ProgramData".TiroObiettivo) AND ("DB320_PID".PID.tiro < 100) THEN
       "DB320_PID".PID.tiro := 1 + "DB320_PID".PID.tiro;
   END_IF;
   IF #_w2 AND ("DB320_PID".PID.tiro > "DB215_ProgramData".TiroObiettivo) THEN
       "DB320_PID".PID.tiro := "DB320_PID".PID.tiro - 1;
   END_IF;
   IF #_w1 THEN "DB215_ProgramData".ContaImpulsi := 1 + "DB215_ProgramData".ContaImpulsi; END_IF;
END_REGION

REGION Network 3: Azzera il contatore ogni 5x (100ms)
   RUNG wire#powerrail
      I_Contact( "On" )
      { S7_Templates := "SrcType := Int" } EQ_Contact(in1 := "DB215_ProgramData".ContaImpulsi, in2 := 4)
      Move(in := 0, out1 => "DB215_ProgramData".ContaImpulsi)
   END_RUNG
   // the same network as SCL:
   IF NOT "On" AND ("DB215_ProgramData".ContaImpulsi = 4) THEN "DB215_ProgramData".ContaImpulsi := 0; END_IF;
END_REGION

REGION Network 4: Impulso ogni 100ms (OB30 x5)
   RUNG wire#powerrail
      I_Contact( "On" )
      { S7_Templates := "SrcType := Int" } EQ_Contact(in1 := "DB215_ProgramData".ContaImpulsi, in2 := 0)
      S_Coil( "BitClock2" )
   END_RUNG
   // the same network as SCL:
   IF NOT "On" AND ("DB215_ProgramData".ContaImpulsi = 0) THEN "BitClock2" := TRUE; END_IF;
END_REGION

REGION Network 5: Impulso ogni 100ms (OB30 x5)
   // Rampa per raggiungere tiro obiettivo e zero, sotto il 20%
   RUNG wire#powerrail
      I_Contact( "On" )
      Contact( "BitClock2" )
      wire#w1
      R_Coil( "BitClock2" )
   END_RUNG
   RUNG wire#w1
      Contact( "Auto" )
      { S7_Templates := "SrcType := Int" } GE_Contact(in1 := "MB0", in2 := 16)
      { S7_Templates := "SrcType := UInt" } LT_Contact(in1 := "DB320_PID".PID.tiro, in2 := 20)
      wire#w2
      { S7_Templates := "SrcType := UInt" } LT_Contact(in1 := "DB320_PID".PID.tiro, in2 := "DB215_ProgramData".TiroObiettivo)
      Add(in1 := 1, in2 := "DB320_PID".PID.tiro, out => "DB320_PID".PID.tiro)
   END_RUNG
   RUNG wire#w2
      { S7_Templates := "SrcType := UInt" } GT_Contact(in1 := "DB320_PID".PID.tiro, in2 := "DB215_ProgramData".TiroObiettivo)
      { S7_Templates := "SrcType := UInt" } GT_Contact(in1 := "DB320_PID".PID.tiro, in2 := 0)
      Sub(in1 := "DB320_PID".PID.tiro, in2 := 1, out => "DB320_PID".PID.tiro)
   END_RUNG
   // the same network as SCL:
   #_w1 := NOT "On" AND "BitClock2";
   IF #_w1 THEN "BitClock2" := FALSE; END_IF;
   #_w2 := #_w1 AND "Auto" AND ("MB0" >= 16) AND ("DB320_PID".PID.tiro < 20);
   IF #_w2 AND ("DB320_PID".PID.tiro < "DB215_ProgramData".TiroObiettivo) THEN
       "DB320_PID".PID.tiro := 1 + "DB320_PID".PID.tiro;
   END_IF;
   IF #_w2 AND ("DB320_PID".PID.tiro > "DB215_ProgramData".TiroObiettivo) AND ("DB320_PID".PID.tiro > 0) THEN
       "DB320_PID".PID.tiro := "DB320_PID".PID.tiro - 1;
   END_IF;
END_REGION

REGION Network 7: Arm rotation and top carriage speed change for DAC M20
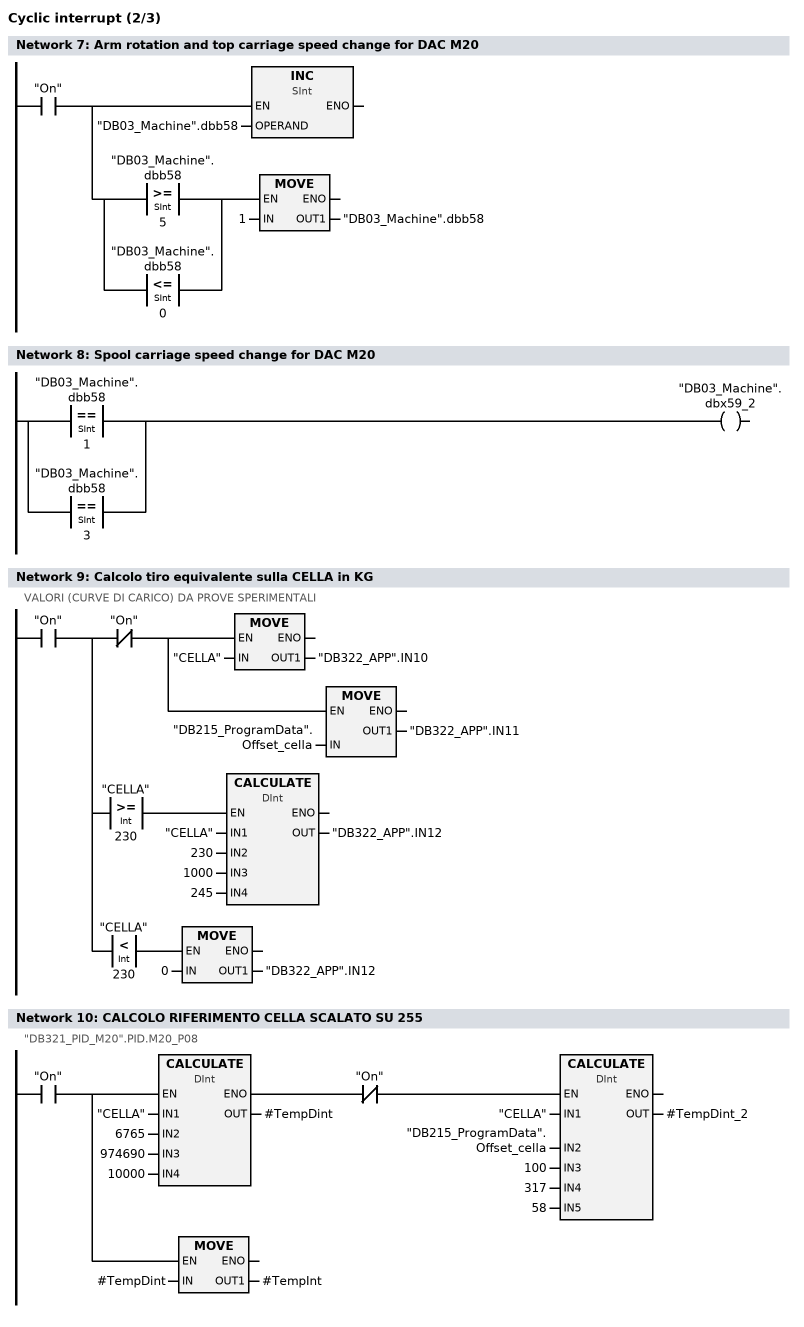
   RUNG wire#powerrail
      Contact( "On" )
      wire#w1
      { S7_Templates := "DestType := SInt"; S7_GenerateENO := "TRUE" } Inc( "DB03_Machine".dbb58 )
   END_RUNG
   RUNG wire#w1
      { S7_Templates := "SrcType := SInt" } GE_Contact(in1 := "DB03_Machine".dbb58, in2 := 5)
      wire#w2
      { S7_GenerateENO := "TRUE" } Move(in := 1, out1 => "DB03_Machine".dbb58)
   END_RUNG
   RUNG wire#w1
      { S7_Templates := "SrcType := SInt" } LE_Contact(in1 := "DB03_Machine".dbb58, in2 := 0)
   END_RUNG wire#w2
   // the same network as SCL:
   IF "On" THEN "DB03_Machine".dbb58 := "DB03_Machine".dbb58 + 1; END_IF;
   IF "On" AND (("DB03_Machine".dbb58 >= 5) OR ("DB03_Machine".dbb58 <= 0)) THEN
       "DB03_Machine".dbb58 := 1;
   END_IF;
END_REGION

REGION Network 8: Spool carriage speed change for DAC M20
   RUNG wire#powerrail
      { S7_Templates := "SrcType := SInt" } EQ_Contact(in1 := "DB03_Machine".dbb58, in2 := 1)
      wire#w1
      Coil( "DB03_Machine".dbx59_2 )
   END_RUNG
   RUNG wire#powerrail
      { S7_Templates := "SrcType := SInt" } EQ_Contact(in1 := "DB03_Machine".dbb58, in2 := 3)
   END_RUNG wire#w1
   // the same network as SCL:
   "DB03_Machine".dbx59_2 := ("DB03_Machine".dbb58 = 1) OR ("DB03_Machine".dbb58 = 3);
END_REGION

REGION Network 9: Calcolo tiro equivalente sulla CELLA in KG
   // VALORI (CURVE DI CARICO) DA PROVE SPERIMENTALI
   RUNG wire#powerrail
      Contact( "On" )
      wire#w1
      I_Contact( "On" )
      wire#w2
      Move(in := "CELLA", out1 => "DB322_APP".IN10)
   END_RUNG
   RUNG wire#w2
      Move(in := "DB215_ProgramData".Offset_cella, out1 => "DB322_APP".IN11)
   END_RUNG
   RUNG wire#w1
      { S7_Templates := "SrcType := Int" } GE_Contact(in1 := "CELLA", in2 := 230)
      { S7_Templates := "SrcType := DInt"; S7_Expression := "((IN1-IN2)*IN3)/IN4" } Calculate(in1 := "CELLA", in2 := 230, in3 := 1000, in4 := 245, out => "DB322_APP".IN12)
   END_RUNG
   RUNG wire#w1
      { S7_Templates := "SrcType := Int" } LT_Contact(in1 := "CELLA", in2 := 230)
      Move(in := 0, out1 => "DB322_APP".IN12)
   END_RUNG
   // the same network as SCL:
   IF "On" AND NOT "On" THEN
       "DB322_APP".IN10 := "CELLA";
       "DB322_APP".IN11 := "DB215_ProgramData".Offset_cella;
   END_IF;
   IF "On" AND ("CELLA" >= 230) THEN "DB322_APP".IN12 := (("CELLA"-230)*1000)/245; END_IF;
   IF "On" AND ("CELLA" < 230) THEN "DB322_APP".IN12 := 0; END_IF;
END_REGION

REGION Network 10: CALCOLO RIFERIMENTO CELLA SCALATO SU 255
   // "DB321_PID_M20".PID.M20_P08
   RUNG wire#powerrail
      Contact( "On" )
      wire#w1
      { S7_Templates := "SrcType := DInt"; S7_Expression := "(IN1*IN2-IN3)/IN4" } Calculate(in1 := "CELLA", in2 := 6765, in3 := 974690, in4 := 10000, out => #TempDint)
      I_Contact( "On" )
      { S7_Templates := "SrcType := DInt"; S7_Expression := "((IN1-IN2)*IN3/IN4)+IN5" } Calculate(in1 := "CELLA", in2 := "DB215_ProgramData".Offset_cella, in3 := 100, in4 := 317, in5 := 58, out => #TempDint_2)
   END_RUNG
   RUNG wire#w1
      Move(in := #TempDint, out1 => #TempInt)
   END_RUNG
   // the same network as SCL:
   IF "On" THEN #TempDint := ("CELLA"*6765-974690)/10000; END_IF;
   IF "On" AND NOT "On" THEN #TempDint_2 := (("CELLA"-"DB215_ProgramData".Offset_cella)*100/317)+58; END_IF;
   IF "On" THEN #TempInt := #TempDint; END_IF;
END_REGION

REGION Network 11: M20
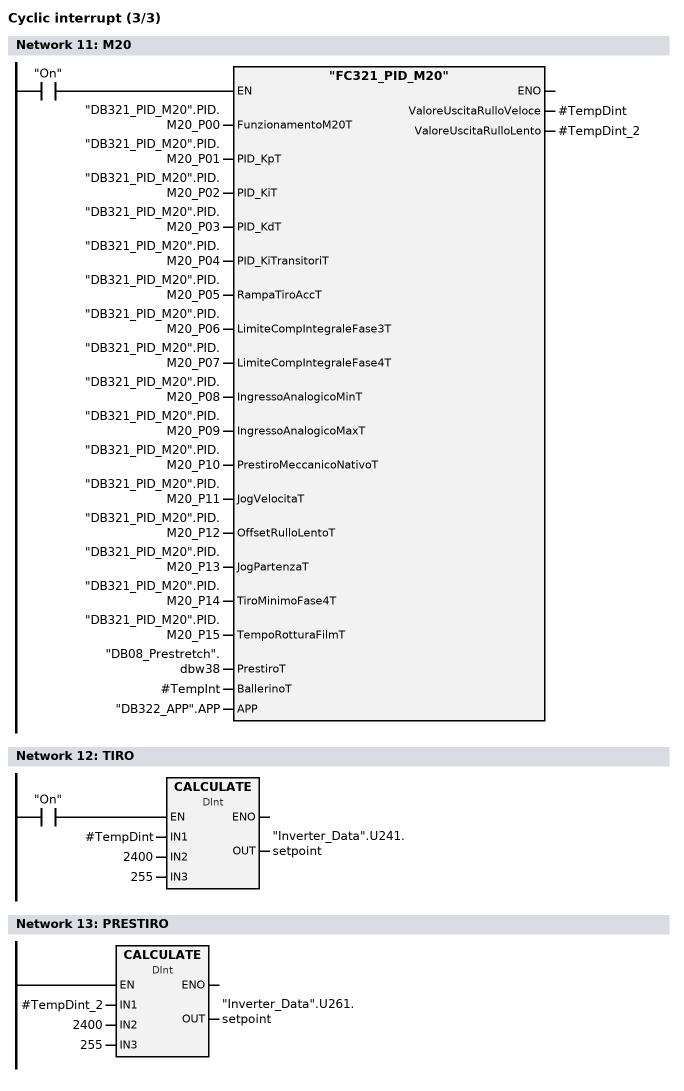
   RUNG wire#powerrail
      Contact( "On" )
      "FC321_PID_M20"(FunzionamentoM20T := "DB321_PID_M20".PID.M20_P00, PID_KpT := "DB321_PID_M20".PID.M20_P01, PID_KiT := "DB321_PID_M20".PID.M20_P02, PID_KdT := "DB321_PID_M20".PID.M20_P03, PID_KiTransitoriT := "DB321_PID_M20".PID.M20_P04, RampaTiroAccT := "DB321_PID_M20".PID.M20_P05, LimiteCompIntegraleFase3T := "DB321_PID_M20".PID.M20_P06, LimiteCompIntegraleFase4T := "DB321_PID_M20".PID.M20_P07, IngressoAnalogicoMinT := "DB321_PID_M20".PID.M20_P08, IngressoAnalogicoMaxT := "DB321_PID_M20".PID.M20_P09, PrestiroMeccanicoNativoT := "DB321_PID_M20".PID.M20_P10, JogVelocitaT := "DB321_PID_M20".PID.M20_P11, OffsetRulloLentoT := "DB321_PID_M20".PID.M20_P12, JogPartenzaT := "DB321_PID_M20".PID.M20_P13, TiroMinimoFase4T := "DB321_PID_M20".PID.M20_P14, TempoRotturaFilmT := "DB321_PID_M20".PID.M20_P15, PrestiroT := "DB08_Prestretch".dbw38, BallerinoT := #TempInt, APP := "DB322_APP".APP, ValoreUscitaRulloVeloce => #TempDint, ValoreUscitaRulloLento => #TempDint_2)
   END_RUNG
   // the same network as SCL:
   IF "On" THEN
       "FC321_PID_M20"(FunzionamentoM20T := "DB321_PID_M20".PID.M20_P00,
                       PID_KpT := "DB321_PID_M20".PID.M20_P01,
                       PID_KiT := "DB321_PID_M20".PID.M20_P02,
                       PID_KdT := "DB321_PID_M20".PID.M20_P03,
                       PID_KiTransitoriT := "DB321_PID_M20".PID.M20_P04,
                       RampaTiroAccT := "DB321_PID_M20".PID.M20_P05,
                       LimiteCompIntegraleFase3T := "DB321_PID_M20".PID.M20_P06,
                       LimiteCompIntegraleFase4T := "DB321_PID_M20".PID.M20_P07,
                       IngressoAnalogicoMinT := "DB321_PID_M20".PID.M20_P08,
                       IngressoAnalogicoMaxT := "DB321_PID_M20".PID.M20_P09,
                       PrestiroMeccanicoNativoT := "DB321_PID_M20".PID.M20_P10,
                       JogVelocitaT := "DB321_PID_M20".PID.M20_P11,
                       OffsetRulloLentoT := "DB321_PID_M20".PID.M20_P12,
                       JogPartenzaT := "DB321_PID_M20".PID.M20_P13,
                       TiroMinimoFase4T := "DB321_PID_M20".PID.M20_P14,
                       TempoRotturaFilmT := "DB321_PID_M20".PID.M20_P15,
                       PrestiroT := "DB08_Prestretch".dbw38,
                       BallerinoT := #TempInt,
                       APP := "DB322_APP".APP,
                       ValoreUscitaRulloVeloce => #TempDint,
                       ValoreUscitaRulloLento => #TempDint_2);
   END_IF;
END_REGION

REGION Network 12: TIRO
   RUNG wire#powerrail
      Contact( "On" )
      { S7_Templates := "SrcType := DInt"; S7_Expression := "IN1*IN2/IN3" } Calculate(in1 := #TempDint, in2 := 2400, in3 := 255, out => "Inverter_Data".U241.setpoint)
   END_RUNG
   // the same network as SCL:
   IF "On" THEN "Inverter_Data".U241.setpoint := #TempDint*2400/255; END_IF;
END_REGION

REGION Network 13: PRESTIRO
   RUNG wire#powerrail
      { S7_Templates := "SrcType := DInt"; S7_Expression := "IN1*IN2/IN3" } Calculate(in1 := #TempDint_2, in2 := 2400, in3 := 255, out => "Inverter_Data".U261.setpoint)
   END_RUNG
   // the same network as SCL:
   "Inverter_Data".U261.setpoint := #TempDint_2*2400/255;
END_REGION
END_ORGANIZATION_BLOCK

FUNCTION "FC321_PID_M20" : Void
{ S7_Optimized_Access := 'TRUE' }
VERSION : 0.1
   VAR_INPUT 
      FunzionamentoM20T : Int;
      PID_KpT : Int;
      PID_KiT : Int;
      PID_KdT : Int;
      PID_KiTransitoriT : Int;
      RampaTiroAccT : Int;
      LimiteCompIntegraleFase3T : Int;
      LimiteCompIntegraleFase4T : Int;
      IngressoAnalogicoMinT : Int;
      IngressoAnalogicoMaxT : Int;
      PrestiroMeccanicoNativoT : Int;
      JogVelocitaT : Int;
      OffsetRulloLentoT : Int;
      JogPartenzaT : Int;
      TiroMinimoFase4T : Int;
      TempoRotturaFilmT : Int;
      PrestiroT : Int;
      BallerinoT : Int;
   END_VAR

   VAR_OUTPUT 
      ValoreUscitaRulloVeloce : DInt;
      ValoreUscitaRulloLento : DInt;
   END_VAR

   VAR_IN_OUT 
      APP : "APP";
   END_VAR

   VAR_TEMP 
      PID_ComponenteProporzionale : DInt;
      PID_ComponenteIntegrale : DInt;
      PID_ComponenteDerivativa : DInt;
      Tiro : Int;
      Tiro1 : Int;
      Tiro2 : Int;
      TiroPrecedente : Int;
      TiroAppoggio : Int;
      ErroreAttuale : Int;
      ErrorePrecedente : Int;
      PID_Kp : Int;
      PID_Ki : Int;
      PID_Kd : Int;
      SetpointTiro : Int;
      SetpointTiroRampa : Int;
      TransitorioInizialeFase1 : Int;
      TransitorioFase3 : Int;
      TransitorioFase4 : Int;
      VelocitaRotazione : Int;
      VelocitaRotazioneFase2 : Int;
      VelocitaRotazioneAppoggio1 : Int;
      VelocitaRotazioneAppoggio2 : Int;
      Fase1OneShoot : Int;
      Fase2OneShoot : Int;
      Fase3OneShoot : Int;
      Fase4OneShoot : Int;
      ArrestoRepentinoOneShoot : Int;
      TiroFase1 : Int;
      TempIntero : Int;
      Fase : Int;
      BallerinoPrecedente : Array[0..2] of Int;
      LimiteComponenteIntegrale : Int;
      TiroRichiesto : Int;
      TimerArrestoRepentino : Int;
      TiroMinimoArrestoRepentino : Int;
      VariazioneTiro : Int;
      TimerFase2 : Int;
      TempoRotturaFilm : Int;
      TimerFase4 : Int;
      TiroMinimoFase4 : Int;
      PID_Uscita : DInt;
      PrestiroRichiesto : DInt;
      PrestiroAppoggio : Real;
   END_VAR

   VAR CONSTANT 
      PID_LimiteSuperioreIntegrale : DInt := 23000;
      PID_LimiteInferioreIntegrale : DInt := 0;
      PID_LimiteSuperioreDerivativa : DInt := 6000;
      PID_LimiteInferioreDerivativa : DInt := -6000;
      PID_LimiteSuperioreUscita : DInt := 255;
      PID_LimiteInferioreUscita : DInt := 0;
   END_VAR


BEGIN
	// Devono esserci due letture uguali per cambiare il valore di tiro. Serve a filtrare letture spurie
	//
	#APP.Tiro1 := "DB08_Prestretch".dbw18; //val_parametro[22];
	//
	IF (#APP.Tiro1 = #APP.Tiro2) THEN
	    #APP.Tiro := #APP.#Tiro1;
	END_IF;
	//
	#APP.Tiro2 := #APP.#Tiro1;
	//
	#APP.VelocitaRotazione := "DB09_TablePos".dbw10; //val_parametro[20];
	//
	// Fase 1:  Accelerazione
	//***********************
	IF (#APP.Tiro = 206) THEN
	    #APP.Fase := 1;
	    //Inizializzazione Fase 1
	    IF (#APP.Fase1OneShoot = 0) THEN
	        #APP.SetpointTiroRampa := #BallerinoT * 10;
	        #APP.TransitorioInizialeFase1 := 1;
	        #APP.Fase1OneShoot := 1;
	        #APP.PID_ComponenteIntegrale := #APP.PID_ComponenteIntegrale + #JogPartenzaT * 100; //Incremento di componente integrale per limitare tiri alti alla partenza 
	    END_IF;
	    //
	    #APP.VariazioneTiro := #BallerinoT - #APP.BallerinoPrecedente[2];
	    //#APP.VariazioneTiro := (#BallerinoT - #APP.BallPrec_2);
	    #APP.PID_Kp := #PID_KpT * 2;
	    #APP.PID_Ki := #PID_KiT * 2;
	    #APP.PID_Kd := #PID_KdT * 3;
	    //
	    IF (#APP.VariazioneTiro < 0) THEN
	        #APP.PID_Kd := 0;
	    END_IF;
	    //
	    IF (#APP.TiroFase1 = 0) THEN
	        #APP.TiroFase1 := 5;
	    END_IF;
	    //
	    #APP.SetpointTiro := ((#IngressoAnalogicoMaxT - #IngressoAnalogicoMinT) * #APP.TiroFase1 / 100) + #IngressoAnalogicoMinT;
	    //
	    //Incremento componente integrale durante la fase di accelerazione per ridurre l'errore sul tiro desiderato
	    IF (#APP.VariazioneTiro > 0 AND #APP.ErroreAttuale > 0) THEN
	        IF (#FunzionamentoM20T = 0) THEN
	            #APP.PID_ComponenteIntegrale := #APP.PID_ComponenteIntegrale + #PID_KpT * #APP.ErroreAttuale / 4;
	        ELSE //(#APP.FunzionamentoM20T == 1)
	            #APP.PID_ComponenteIntegrale := #APP.PID_ComponenteIntegrale + #PID_KpT * #APP.ErroreAttuale / 10;
	        END_IF;
	    END_IF;
	    //Rampa di tiro per tiri alti
	    IF (#APP.TransitorioInizialeFase1 = 1) THEN
	        IF (#APP.SetpointTiroRampa / 10 < #APP.SetpointTiro) THEN
	            #APP.SetpointTiroRampa := #APP.SetpointTiroRampa + #RampaTiroAccT;
	            #APP.SetpointTiro := #APP.SetpointTiroRampa / 10;
	        ELSE
	            #APP.TransitorioInizialeFase1 := 0;
	        END_IF;
	    END_IF;
	    #APP.TiroRichiesto := #APP.TiroFase1;
	END_IF;
	//
	// Fase 2: Fasciatura a regime
	//****************************
	IF (#APP.Tiro > 0 AND #APP.Tiro <= 100) THEN
	    #APP.Fase := 2;
	    #APP.Fase4OneShoot := 0;
	    // Inizializzazione Fase 2      
	    IF (#APP.Fase2OneShoot = 0) THEN
	        #APP.VelocitaRotazioneFase2 := 0;
	        #APP.Fase2OneShoot := 1;
	        // PID_ComponenteIntegrale = PID_ComponenteIntegrale+2000; //Fornisco un piccolo delta di velocita'alla partenza per evitare di tirare strattoni sul ballerino all'avvio 
	    END_IF;
	    #APP.PID_Kp := #PID_KpT;
	    #APP.PID_Ki := #PID_KiT;
	    #APP.PID_Kd := #PID_KdT;
	    IF (#APP.Tiro >= 50) THEN
	        #APP.PID_Ki := (15 + 20 * #PID_KiT) / 30; //Per tiri alti diminuisco il guadagno integrale per rendere il regolatore meno pronto e farlo oscillare meno.
	    END_IF;
	    #APP.SetpointTiro := ((#IngressoAnalogicoMaxT - #IngressoAnalogicoMinT) * #APP.Tiro / 100) + #IngressoAnalogicoMinT;
	    #APP.TiroFase1 := #APP.Tiro;
	    //
	    //Velocita' di rotazione braccio nella Fase 2. Filtro di 3 scansioni
	    IF (#APP.VelocitaRotazione = #APP.VelocitaRotazioneAppoggio1 AND #APP.VelocitaRotazioneAppoggio1 = #APP.VelocitaRotazioneAppoggio2) THEN
	        #APP.VelocitaRotazioneFase2 := #APP.VelocitaRotazione;
	    END_IF;
	    #APP.VelocitaRotazioneAppoggio2 := #APP.VelocitaRotazioneAppoggio1;
	    #APP.VelocitaRotazioneAppoggio1 := #APP.VelocitaRotazione;
	    //
	    //Rottura film
	    IF (#BallerinoT < #IngressoAnalogicoMinT) THEN
	        #APP.TimerFase2 := #APP.TimerFase2 + 1;
	    ELSE
	        #APP.TimerFase2 := 0;
	    END_IF;
	    //
	    #APP.TempoRotturaFilm := #TempoRotturaFilmT * 10 / 3; //Tempo rottura film in numero di scansioni
	    IF (#APP.TimerFase2 >= #APP.TempoRotturaFilm) THEN
	        #APP.PID_ComponenteIntegrale := 0;
	        #APP.TimerFase2 := 0;
	    END_IF;
	    #APP.TiroRichiesto := #APP.Tiro;
	END_IF;
	//
	// Fase 3: Transitorio velocita' alta -> media
	//********************************************
	IF (#APP.Tiro > 100 AND #APP.Tiro <= 200) THEN
	    #APP.Fase := 3;
	    #APP.Fase4OneShoot := 0;
	    //
	    // Inizializzazione Fase 3
	    IF (#APP.Fase3OneShoot = 0) THEN
	        #APP.TransitorioFase3 := 0;
	        #APP.Fase3OneShoot := 1;
	    END_IF;
	    //
	    #APP.LimiteComponenteIntegrale := #LimiteCompIntegraleFase3T * 100;
	    #APP.PID_Kp := #PID_KpT;
	    #APP.PID_Ki := #PID_KiTransitoriT;
	    #APP.PID_Kd := #PID_KdT;
	    #APP.SetpointTiro := ((#IngressoAnalogicoMaxT - #IngressoAnalogicoMinT) * (#APP.Tiro - 100) / 100) + #IngressoAnalogicoMinT;
	    //
	    #APP.TempIntero := #APP.VelocitaRotazioneFase2 * 9 / 10;
	    IF (#APP.VelocitaRotazione < #APP.TempIntero AND #APP.TransitorioFase3 = 0) THEN
	        #APP.TransitorioFase3 := 1;
	        IF (#APP.PID_ComponenteIntegrale > #APP.LimiteComponenteIntegrale) THEN
	            #APP.PID_ComponenteIntegrale := #APP.LimiteComponenteIntegrale;
	        END_IF;
	    END_IF;
	    #APP.TiroRichiesto := #APP.Tiro - 100;
	END_IF;
	//
	// Fase 4: Transitorio velocita' media -> bassa
	// ********************************************
	IF (#APP.Tiro = 201) THEN
	    #APP.Fase := 4;
	    // Inizializzazione Fase 4
	    IF (#APP.Fase4OneShoot = 0) THEN
	        #APP.TransitorioFase4 := 0;
	        #APP.Fase4OneShoot := 1;
	    END_IF;
	    //
	    IF (#APP.TiroPrecedente <= 100) THEN
	        #APP.TiroAppoggio := #APP.TiroPrecedente;
	    END_IF;
	    //
	    IF (#APP.TiroPrecedente > 100 AND #APP.TiroPrecedente <= 200) THEN
	        #APP.TiroAppoggio := #APP.TiroPrecedente - 100;
	    END_IF;
	    //
	    //Alzo il tiro richiesto nei primi decimi, in maniera da abbattere la componente integrale
	    #APP.TiroMinimoFase4 := #TiroMinimoFase4T;
	    //
	    IF (#APP.TiroAppoggio < #APP.TiroMinimoFase4) THEN
	        #APP.TiroAppoggio := #APP.TiroMinimoFase4;
	    END_IF;
	    //
	    #APP.SetpointTiro := ((#IngressoAnalogicoMaxT - #IngressoAnalogicoMinT) * #APP.TiroAppoggio / 100) + #IngressoAnalogicoMinT;
	    //
	    #APP.LimiteComponenteIntegrale := #LimiteCompIntegraleFase4T * 100;
	    #APP.PID_Kp := #PID_KpT;
	    #APP.PID_Ki := #PID_KiTransitoriT * 15 / 10;
	    #APP.PID_Kd := #PID_KdT;
	    IF (#APP.PID_ComponenteIntegrale > #APP.LimiteComponenteIntegrale) THEN
	        #APP.PID_ComponenteIntegrale := #APP.LimiteComponenteIntegrale;
	    END_IF;
	    //
	    #APP.TransitorioFase4 := 1;
	    #APP.TiroRichiesto := #APP.TiroAppoggio;
	END_IF;
	//
	// Fase 0: Azzeramento del regolatore
	// **********************************
	IF (#APP.Tiro = 0) THEN
	    #APP.Fase := 0;
	    #APP.PID_ComponenteIntegrale := 0;
	    #APP.Fase1OneShoot := 0;
	    #APP.Fase2OneShoot := 0;
	    #APP.Fase3OneShoot := 0;
	    #APP.Fase4OneShoot := 0;
	    #APP.ArrestoRepentinoOneShoot := 0;
	    #APP.SetpointTiro := #BallerinoT;
	    #APP.TiroPrecedente := 0;
	    #APP.TiroFase1 := 0;
	    #APP.TiroAppoggio := 0;
	END_IF;
	//   
	// Jog in manuale
	// **************
	IF (#APP.Tiro = 210) THEN
	    #APP.PID_Kp := 0;
	    #APP.PID_Ki := 0;
	    #APP.PID_Kd := 0;
	    #APP.PID_ComponenteIntegrale := #JogVelocitaT * 100;
	END_IF;
	//   
	// Arresto repentino
	// *****************
	IF (#APP.Tiro = 202) THEN
	    // Inizializzazione Fase 4
	    IF (#APP.ArrestoRepentinoOneShoot = 0) THEN
	        #APP.TimerArrestoRepentino := 0;
	        #APP.ArrestoRepentinoOneShoot := 1;
	    END_IF;
	    //
	    #APP.TimerArrestoRepentino := #APP.TimerArrestoRepentino + 1;
	    #APP.TiroMinimoArrestoRepentino := #TiroMinimoFase4T * 175 / 100;
	    //
	    IF (#APP.TiroPrecedente <= 100) THEN
	        #APP.TiroAppoggio := #APP.TiroPrecedente;
	    END_IF;
	    //
	    IF (#APP.TiroPrecedente > 100 & #APP.TiroPrecedente <= 200) THEN
	        #APP.TiroAppoggio := #APP.TiroPrecedente - 100;
	    END_IF;
	    //
	    IF (#APP.TiroAppoggio < #APP.TiroMinimoArrestoRepentino) THEN
	        #APP.TiroAppoggio := #APP.TiroMinimoArrestoRepentino;
	    END_IF;
	    //
	    #APP.SetpointTiro := ((#IngressoAnalogicoMaxT - #IngressoAnalogicoMinT) * #APP.TiroAppoggio / 100) + #IngressoAnalogicoMinT;
	    //   
	    #APP.PID_Kp := #PID_KpT;
	    #APP.PID_Ki := #PID_KiTransitoriT * 175 / 100;
	    #APP.PID_Kd := #PID_KdT;
	    //
	    #APP.TiroRichiesto := #APP.TiroAppoggio;
	END_IF;
	//
	// Regolatore PID standard 
	#APP.ErroreAttuale := (#BallerinoT - #APP.SetpointTiro);
	//
	// Componente proporzionale del regolatore          
	#APP.PID_ComponenteProporzionale := #APP.PID_Kp * #APP.ErroreAttuale;
	//
	// Componente integrale del regolatore
	#APP.PID_ComponenteIntegrale := #APP.PID_ComponenteIntegrale + #APP.PID_Ki * #APP.ErroreAttuale / 10;
	//
	IF (#APP.PID_ComponenteIntegrale > #PID_LimiteSuperioreIntegrale AND #APP.Tiro <> 210) THEN
	    #APP.PID_ComponenteIntegrale := #PID_LimiteSuperioreIntegrale;
	END_IF;
	//
	IF (#APP.PID_ComponenteIntegrale > 25500 AND #APP.Tiro = 210) THEN
	    #APP.PID_ComponenteIntegrale := 25500;
	END_IF;
	//
	IF (#APP.PID_ComponenteIntegrale < #PID_LimiteInferioreIntegrale) THEN
	    #APP.PID_ComponenteIntegrale := #PID_LimiteInferioreIntegrale;
	END_IF;
	//
	// Componente derivativa del regolatore
	// PID_ComponenteDerivativa = 10*PID_Kd*(ErroreAttuale-ErrorePrecedente);
	
	#APP.PID_ComponenteDerivativa := 10 * #APP.PID_Kd * (#BallerinoT - #APP.BallerinoPrecedente[2]);
	
	//#PID_ComponenteDerivativa := 10 * #PID_Kd * (#BallerinoT - #APP.BallPrec_2);
	//
	IF (#APP.PID_ComponenteDerivativa > #PID_LimiteSuperioreDerivativa) THEN
	    #APP.PID_ComponenteDerivativa := #PID_LimiteSuperioreDerivativa;
	END_IF;
	//
	IF (#APP.PID_ComponenteDerivativa < #PID_LimiteInferioreDerivativa) THEN
	    #APP.PID_ComponenteDerivativa := #PID_LimiteInferioreDerivativa;
	END_IF;
	//
	#APP.PID_Uscita := (#APP.PID_ComponenteProporzionale + #APP.PID_ComponenteIntegrale + #APP.PID_ComponenteDerivativa) / 100; //Le costanti Kp, Ki e Kd sono espresse nel display in centesimi
	//
	IF (#APP.PID_Uscita > #PID_LimiteSuperioreUscita) THEN
	    #APP.PID_Uscita := #PID_LimiteSuperioreUscita;
	END_IF;
	//
	IF (#APP.PID_Uscita < #PID_LimiteInferioreUscita) THEN
	    #APP.PID_Uscita := #PID_LimiteInferioreUscita;
	END_IF;
	//
	IF (#APP.Tiro = 0) THEN
	    #APP.PID_Uscita := 0;
	END_IF;
	//
	// Aggiornamento valori precedenti  
	#APP.ErrorePrecedente := #APP.ErroreAttuale;
	//
	IF (#APP.Tiro <= 200) THEN
	    #APP.TiroPrecedente := #APP.Tiro;
	END_IF;
	//
	#APP.BallerinoPrecedente[2] := #APP.BallerinoPrecedente[1];
	#APP.BallerinoPrecedente[1] := #APP.BallerinoPrecedente[0];
	#APP.BallerinoPrecedente[0] := #BallerinoT;
	// #APP.BallPrec_2 := #APP.BallPrec_1;
	// #APP.BallPrec_1 := #APP.BallPrec_0;
	// #APP.BallPrec_0 := #BallerinoT;
	//
	// Attuazione delle uscite analogiche che vanno agli inverter
	#ValoreUscitaRulloVeloce := #APP.PID_Uscita;
	
	// Prestiro per PGSM e PGSA
	IF (#FunzionamentoM20T = 0) THEN
	    //
	    #APP.PrestiroRichiesto := INT_TO_DINT(#PrestiroT) * 500 / 255 + 100;
	    // Arrotonda sempre all'intero inferiore, a prescindere. Sommando 0.5 arrotondo all'intero piu vicino
	    #APP.PrestiroAppoggio := 0.5 + DINT_TO_REAL(#ValoreUscitaRulloVeloce * (#PrestiroMeccanicoNativoT + 100) / #APP.PrestiroRichiesto);
	    #APP.PrestiroAppoggio := #APP.PrestiroAppoggio + (#OffsetRulloLentoT - 10);
	    IF (#APP.PrestiroAppoggio > 255) THEN
	        #APP.PrestiroAppoggio := 255;
	    END_IF;
	    #ValoreUscitaRulloLento := REAL_TO_DINT(#APP.PrestiroAppoggio);
	END_IF;
	//
	// Tiro ballerino SCSP valvola proporzionale        
	IF (#FunzionamentoM20T = 1) THEN
	    #ValoreUscitaRulloLento := #PrestiroT;
	    IF (#ValoreUscitaRulloLento > 255) THEN
	        #ValoreUscitaRulloLento := 255;
	    END_IF;
	END_IF;
	
	
	
END_FUNCTION

FUNCTION "FUNÇAO" : Void   // FC1, LAD
{ S7_Optimized_Access := 'TRUE' }
VERSION : 0.1
// stored: AutoNumber true, IsIECCheckEnabled false, SetENOAutomatically false, UDAEnableTagReadback false
BEGIN

REGION Network 1
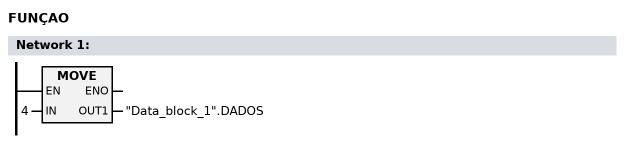
   RUNG wire#powerrail
      Move(in := 4, out1 => "Data_block_1".DADOS)
   END_RUNG
   // the same network as SCL:
   "Data_block_1".DADOS := 4;
END_REGION
END_FUNCTION

FUNCTION "Denormalisation" : Void   // FC14, FBD
{ S7_Optimized_Access := 'TRUE' }
VERSION : 0.1
// stored: AutoNumber true, IsIECCheckEnabled false, SetENOAutomatically false, UDAEnableTagReadback false
   VAR_INPUT
      actual_value_INT : Int;
      normalisation : Real;
   END_VAR
   VAR_OUTPUT
      actual_value_REAL : Real;
   END_VAR
   VAR_TEMP
      temp_actual_value_DINT : DInt;
      temp_actual_value_REAL : Real;
   END_VAR
BEGIN

REGION Network 1
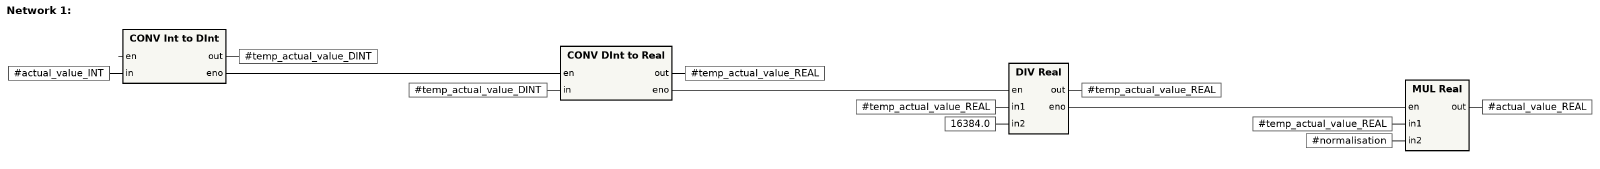
   // ENO of a box is taken as its EN; it also drops when the box reports an error
   #temp_actual_value_DINT := INT_TO_DINT(#actual_value_INT);
   #temp_actual_value_REAL := DINT_TO_REAL(#temp_actual_value_DINT);
   #temp_actual_value_REAL := #temp_actual_value_REAL / 16384.0;
   #actual_value_REAL := #temp_actual_value_REAL * #normalisation;
END_REGION
END_FUNCTION

FUNCTION "FC01_SupportOut" : Void   // FC1, LAD
TITLE = Output support memory
{ S7_Optimized_Access := 'FALSE' }
AUTHOR : Robopac
VERSION : 0.0
// stored: AutoNumber false, IsIECCheckEnabled false, SetENOAutomatically false, UDAEnableTagReadback false
BEGIN

REGION Network 1: STANDARD
END_REGION

REGION Network 2: Emergency mode lamp (Technoplat)
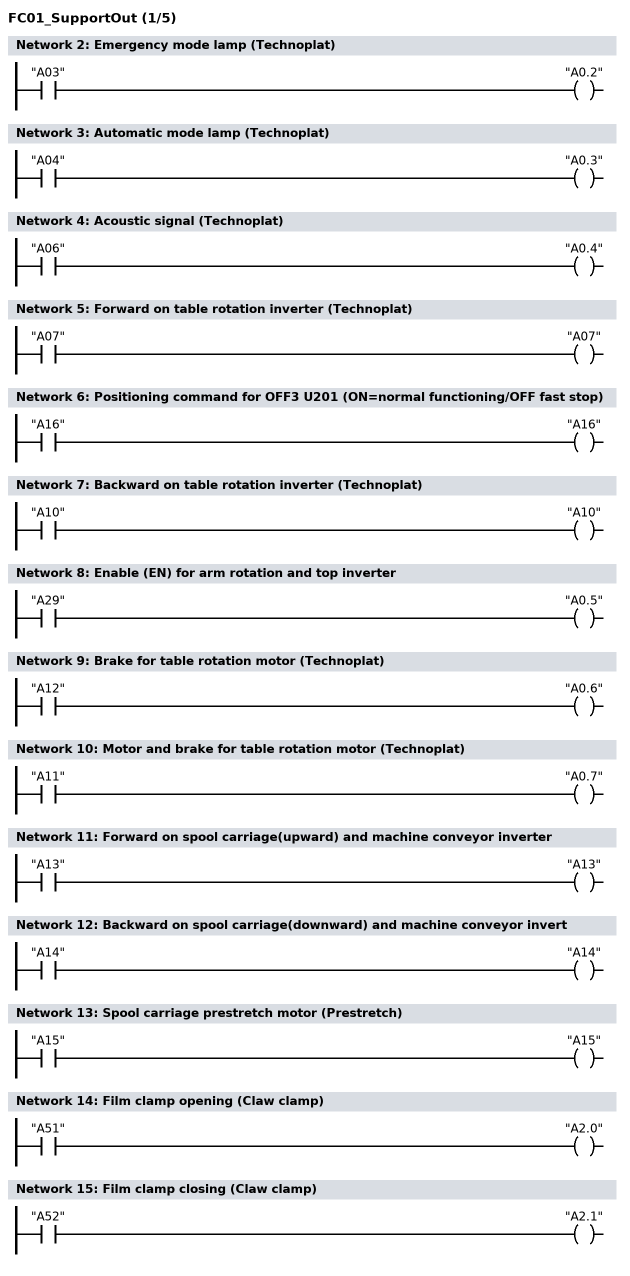
   RUNG wire#powerrail
      Contact( "A03" )
      Coil( "A0.2" )
   END_RUNG
   // the same network as SCL:
   "A0.2" := "A03";
END_REGION

REGION Network 3: Automatic mode lamp (Technoplat)
   RUNG wire#powerrail
      Contact( "A04" )
      Coil( "A0.3" )
   END_RUNG
   // the same network as SCL:
   "A0.3" := "A04";
END_REGION

REGION Network 4: Acoustic signal (Technoplat)
   RUNG wire#powerrail
      Contact( "A06" )
      Coil( "A0.4" )
   END_RUNG
   // the same network as SCL:
   "A0.4" := "A06";
END_REGION

REGION Network 5: Forward on table rotation inverter (Technoplat)
   RUNG wire#powerrail
      Contact( "A07" )
      Coil( "A07" )
   END_RUNG
   // the same network as SCL:
   "A07" := "A07";
END_REGION

REGION Network 6: Positioning command for OFF3 U201 (ON=normal functioning/OFF fast stop)
   RUNG wire#powerrail
      Contact( "A16" )
      Coil( "A16" )
   END_RUNG
   // the same network as SCL:
   "A16" := "A16";
END_REGION

REGION Network 7: Backward on table rotation inverter (Technoplat)
   RUNG wire#powerrail
      Contact( "A10" )
      Coil( "A10" )
   END_RUNG
   // the same network as SCL:
   "A10" := "A10";
END_REGION

REGION Network 8: Enable (EN) for arm rotation and top inverter
   RUNG wire#powerrail
      Contact( "A29" )
      Coil( "A0.5" )
   END_RUNG
   // the same network as SCL:
   "A0.5" := "A29";
END_REGION

REGION Network 9: Brake for table rotation motor (Technoplat)
   RUNG wire#powerrail
      Contact( "A12" )
      Coil( "A0.6" )
   END_RUNG
   // the same network as SCL:
   "A0.6" := "A12";
END_REGION

REGION Network 10: Motor and brake for table rotation motor (Technoplat)
   RUNG wire#powerrail
      Contact( "A11" )
      Coil( "A0.7" )
   END_RUNG
   // the same network as SCL:
   "A0.7" := "A11";
END_REGION

REGION Network 11: Forward on spool carriage(upward) and machine conveyor inverter
   RUNG wire#powerrail
      Contact( "A13" )
      Coil( "A13" )
   END_RUNG
   // the same network as SCL:
   "A13" := "A13";
END_REGION

REGION Network 12: Backward on spool carriage(downward) and machine conveyor invert
   RUNG wire#powerrail
      Contact( "A14" )
      Coil( "A14" )
   END_RUNG
   // the same network as SCL:
   "A14" := "A14";
END_REGION

REGION Network 13: Spool carriage prestretch motor (Prestretch)
   RUNG wire#powerrail
      Contact( "A15" )
      Coil( "A15" )
   END_RUNG
   // the same network as SCL:
   "A15" := "A15";
END_REGION

REGION Network 14: Film clamp opening (Claw clamp)
   RUNG wire#powerrail
      Contact( "A51" )
      Coil( "A2.0" )
   END_RUNG
   // the same network as SCL:
   "A2.0" := "A51";
END_REGION

REGION Network 15: Film clamp closing (Claw clamp)
   RUNG wire#powerrail
      Contact( "A52" )
      Coil( "A2.1" )
   END_RUNG
   // the same network as SCL:
   "A2.1" := "A52";
END_REGION

REGION Network 16: Cutting and welding unit forward(1)/backward (Claw clamp)
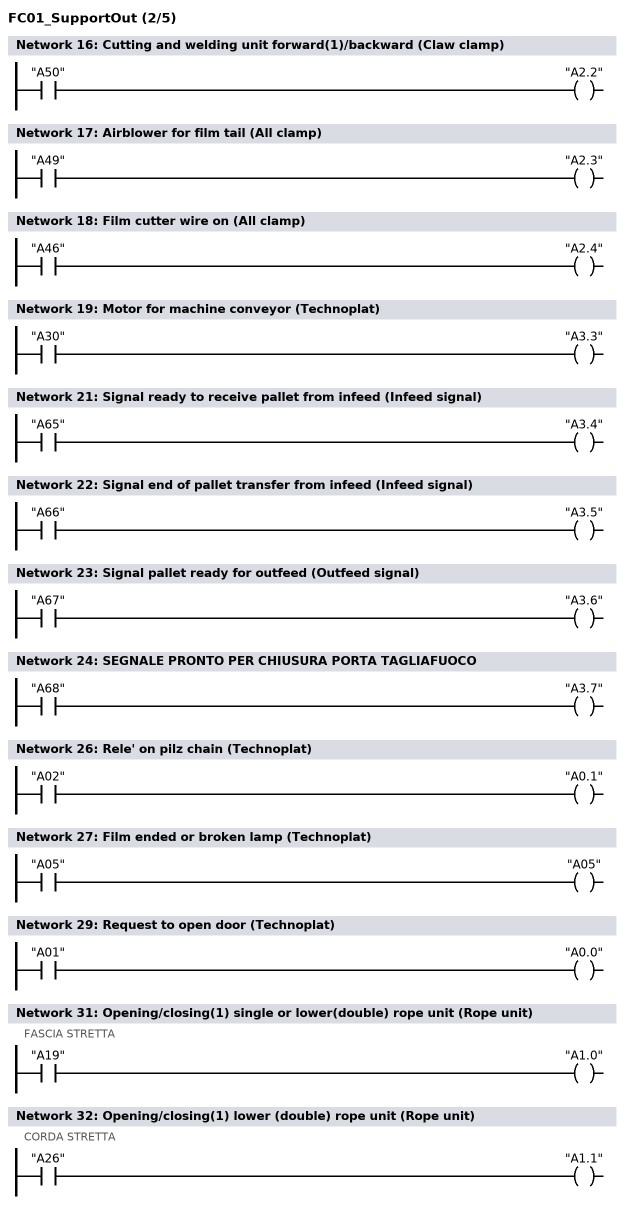
   RUNG wire#powerrail
      Contact( "A50" )
      Coil( "A2.2" )
   END_RUNG
   // the same network as SCL:
   "A2.2" := "A50";
END_REGION

REGION Network 17: Airblower for film tail (All clamp)
   RUNG wire#powerrail
      Contact( "A49" )
      Coil( "A2.3" )
   END_RUNG
   // the same network as SCL:
   "A2.3" := "A49";
END_REGION

REGION Network 18: Film cutter wire on (All clamp)
   RUNG wire#powerrail
      Contact( "A46" )
      Coil( "A2.4" )
   END_RUNG
   // the same network as SCL:
   "A2.4" := "A46";
END_REGION

REGION Network 19: Motor for machine conveyor (Technoplat)
   RUNG wire#powerrail
      Contact( "A30" )
      Coil( "A3.3" )
   END_RUNG
   // the same network as SCL:
   "A3.3" := "A30";
END_REGION

REGION Network 20: EXCHANGE SIGNALS
END_REGION

REGION Network 21: Signal ready to receive pallet from infeed (Infeed signal)
   RUNG wire#powerrail
      Contact( "A65" )
      Coil( "A3.4" )
   END_RUNG
   // the same network as SCL:
   "A3.4" := "A65";
END_REGION

REGION Network 22: Signal end of pallet transfer from infeed (Infeed signal)
   RUNG wire#powerrail
      Contact( "A66" )
      Coil( "A3.5" )
   END_RUNG
   // the same network as SCL:
   "A3.5" := "A66";
END_REGION

REGION Network 23: Signal pallet ready for outfeed (Outfeed signal)
   RUNG wire#powerrail
      Contact( "A67" )
      Coil( "A3.6" )
   END_RUNG
   // the same network as SCL:
   "A3.6" := "A67";
END_REGION

REGION Network 24: SEGNALE PRONTO PER CHIUSURA PORTA TAGLIAFUOCO
   RUNG wire#powerrail
      Contact( "A68" )
      Coil( "A3.7" )
   END_RUNG
   // the same network as SCL:
   "A3.7" := "A68";
END_REGION

REGION Network 25: ACCESSORIES
END_REGION

REGION Network 26: Rele' on pilz chain (Technoplat)
   RUNG wire#powerrail
      Contact( "A02" )
      Coil( "A0.1" )
   END_RUNG
   // the same network as SCL:
   "A0.1" := "A02";
END_REGION

REGION Network 27: Film ended or broken lamp (Technoplat)
   RUNG wire#powerrail
      Contact( "A05" )
      Coil( "A05" )
   END_RUNG
   // the same network as SCL:
   "A05" := "A05";
END_REGION

REGION Network 28: ***DOOR***
END_REGION

REGION Network 29: Request to open door (Technoplat)
   RUNG wire#powerrail
      Contact( "A01" )
      Coil( "A0.0" )
   END_RUNG
   // the same network as SCL:
   "A0.0" := "A01";
END_REGION

REGION Network 30: ***BAND/ROPE***
END_REGION

REGION Network 31: Opening/closing(1) single or lower(double) rope unit (Rope unit)
   // FASCIA STRETTA
   RUNG wire#powerrail
      Contact( "A19" )
      Coil( "A1.0" )
   END_RUNG
   // the same network as SCL:
   "A1.0" := "A19";
END_REGION

REGION Network 32: Opening/closing(1) lower (double) rope unit (Rope unit)
   // CORDA STRETTA
   RUNG wire#powerrail
      Contact( "A26" )
      Coil( "A1.1" )
   END_RUNG
   // the same network as SCL:
   "A1.1" := "A26";
END_REGION

REGION Network 33: ***WELDER***
END_REGION

REGION Network 34: Film welder on (All clamp)
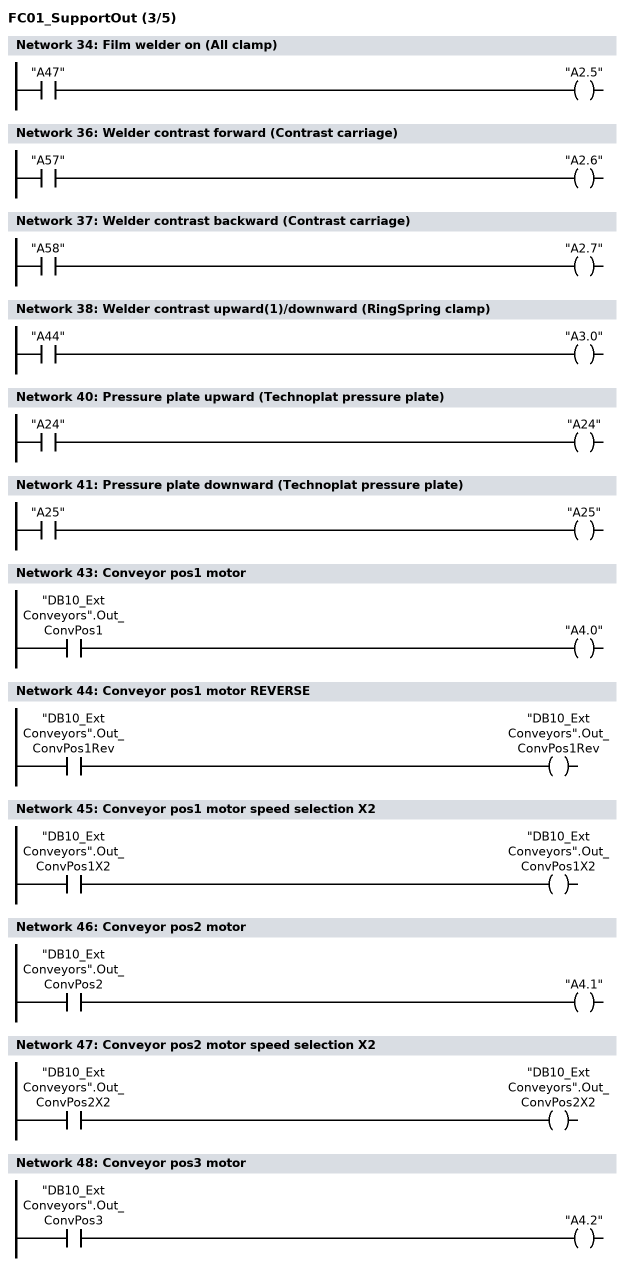
   RUNG wire#powerrail
      Contact( "A47" )
      Coil( "A2.5" )
   END_RUNG
   // the same network as SCL:
   "A2.5" := "A47";
END_REGION

REGION Network 35: ***CONTRAST***
END_REGION

REGION Network 36: Welder contrast forward (Contrast carriage)
   RUNG wire#powerrail
      Contact( "A57" )
      Coil( "A2.6" )
   END_RUNG
   // the same network as SCL:
   "A2.6" := "A57";
END_REGION

REGION Network 37: Welder contrast backward (Contrast carriage)
   RUNG wire#powerrail
      Contact( "A58" )
      Coil( "A2.7" )
   END_RUNG
   // the same network as SCL:
   "A2.7" := "A58";
END_REGION

REGION Network 38: Welder contrast upward(1)/downward (RingSpring clamp)
   RUNG wire#powerrail
      Contact( "A44" )
      Coil( "A3.0" )
   END_RUNG
   // the same network as SCL:
   "A3.0" := "A44";
END_REGION

REGION Network 39: ***PRESSURE***
END_REGION

REGION Network 40: Pressure plate upward (Technoplat pressure plate)
   RUNG wire#powerrail
      Contact( "A24" )
      Coil( "A24" )
   END_RUNG
   // the same network as SCL:
   "A24" := "A24";
END_REGION

REGION Network 41: Pressure plate downward (Technoplat pressure plate)
   RUNG wire#powerrail
      Contact( "A25" )
      Coil( "A25" )
   END_RUNG
   // the same network as SCL:
   "A25" := "A25";
END_REGION

REGION Network 42: ***CONVEYORS***
END_REGION

REGION Network 43: Conveyor pos1 motor
   RUNG wire#powerrail
      Contact( "DB10_ExtConveyors".Out_ConvPos1 )
      Coil( "A4.0" )
   END_RUNG
   // the same network as SCL:
   "A4.0" := "DB10_ExtConveyors".Out_ConvPos1;
END_REGION

REGION Network 44: Conveyor pos1 motor REVERSE
   RUNG wire#powerrail
      Contact( "DB10_ExtConveyors".Out_ConvPos1Rev )
      Coil( "DB10_ExtConveyors".Out_ConvPos1Rev )
   END_RUNG
   // the same network as SCL:
   "DB10_ExtConveyors".Out_ConvPos1Rev := "DB10_ExtConveyors".Out_ConvPos1Rev;
END_REGION

REGION Network 45: Conveyor pos1 motor speed selection X2
   RUNG wire#powerrail
      Contact( "DB10_ExtConveyors".Out_ConvPos1X2 )
      Coil( "DB10_ExtConveyors".Out_ConvPos1X2 )
   END_RUNG
   // the same network as SCL:
   "DB10_ExtConveyors".Out_ConvPos1X2 := "DB10_ExtConveyors".Out_ConvPos1X2;
END_REGION

REGION Network 46: Conveyor pos2 motor
   RUNG wire#powerrail
      Contact( "DB10_ExtConveyors".Out_ConvPos2 )
      Coil( "A4.1" )
   END_RUNG
   // the same network as SCL:
   "A4.1" := "DB10_ExtConveyors".Out_ConvPos2;
END_REGION

REGION Network 47: Conveyor pos2 motor speed selection X2
   RUNG wire#powerrail
      Contact( "DB10_ExtConveyors".Out_ConvPos2X2 )
      Coil( "DB10_ExtConveyors".Out_ConvPos2X2 )
   END_RUNG
   // the same network as SCL:
   "DB10_ExtConveyors".Out_ConvPos2X2 := "DB10_ExtConveyors".Out_ConvPos2X2;
END_REGION

REGION Network 48: Conveyor pos3 motor
   RUNG wire#powerrail
      Contact( "DB10_ExtConveyors".Out_ConvPos3 )
      Coil( "A4.2" )
   END_RUNG
   // the same network as SCL:
   "A4.2" := "DB10_ExtConveyors".Out_ConvPos3;
END_REGION

REGION Network 49: Conveyor pos4 motor
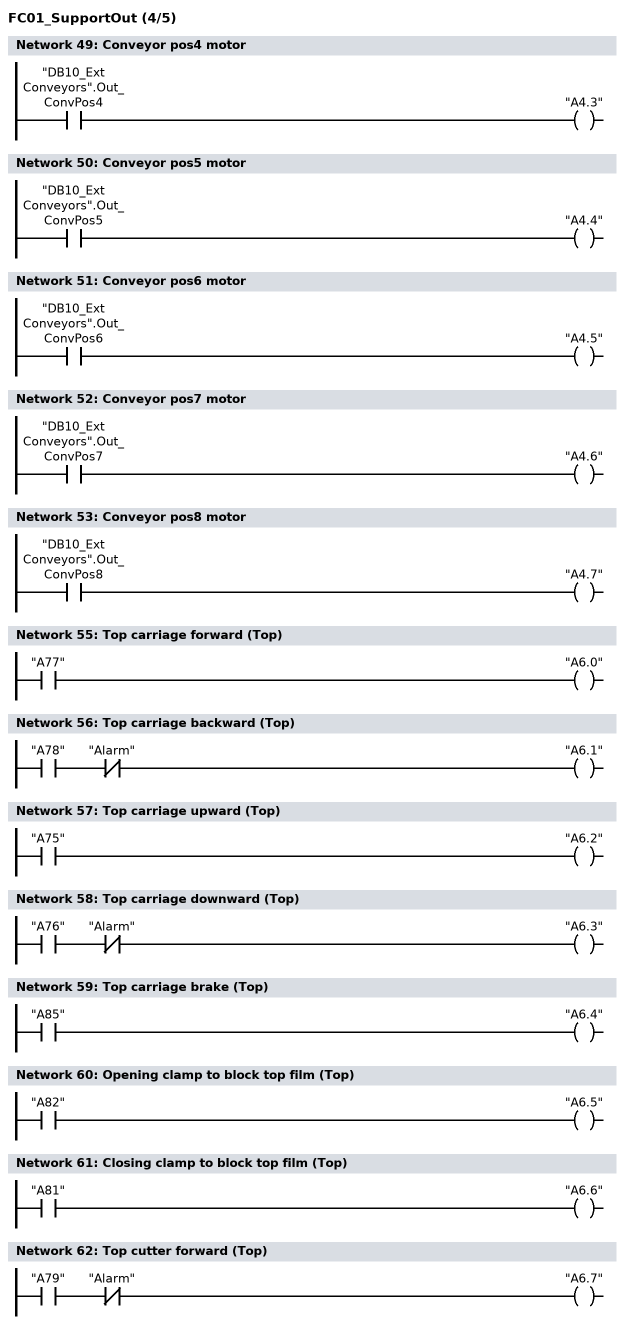
   RUNG wire#powerrail
      Contact( "DB10_ExtConveyors".Out_ConvPos4 )
      Coil( "A4.3" )
   END_RUNG
   // the same network as SCL:
   "A4.3" := "DB10_ExtConveyors".Out_ConvPos4;
END_REGION

REGION Network 50: Conveyor pos5 motor
   RUNG wire#powerrail
      Contact( "DB10_ExtConveyors".Out_ConvPos5 )
      Coil( "A4.4" )
   END_RUNG
   // the same network as SCL:
   "A4.4" := "DB10_ExtConveyors".Out_ConvPos5;
END_REGION

REGION Network 51: Conveyor pos6 motor
   RUNG wire#powerrail
      Contact( "DB10_ExtConveyors".Out_ConvPos6 )
      Coil( "A4.5" )
   END_RUNG
   // the same network as SCL:
   "A4.5" := "DB10_ExtConveyors".Out_ConvPos6;
END_REGION

REGION Network 52: Conveyor pos7 motor
   RUNG wire#powerrail
      Contact( "DB10_ExtConveyors".Out_ConvPos7 )
      Coil( "A4.6" )
   END_RUNG
   // the same network as SCL:
   "A4.6" := "DB10_ExtConveyors".Out_ConvPos7;
END_REGION

REGION Network 53: Conveyor pos8 motor
   RUNG wire#powerrail
      Contact( "DB10_ExtConveyors".Out_ConvPos8 )
      Coil( "A4.7" )
   END_RUNG
   // the same network as SCL:
   "A4.7" := "DB10_ExtConveyors".Out_ConvPos8;
END_REGION

REGION Network 54: ***TOP***
END_REGION

REGION Network 55: Top carriage forward (Top)
   RUNG wire#powerrail
      Contact( "A77" )
      Coil( "A6.0" )
   END_RUNG
   // the same network as SCL:
   "A6.0" := "A77";
END_REGION

REGION Network 56: Top carriage backward (Top)
   RUNG wire#powerrail
      Contact( "A78" )
      I_Contact( "Alarm" )
      Coil( "A6.1" )
   END_RUNG
   // the same network as SCL:
   "A6.1" := "A78" AND NOT "Alarm";
END_REGION

REGION Network 57: Top carriage upward (Top)
   RUNG wire#powerrail
      Contact( "A75" )
      Coil( "A6.2" )
   END_RUNG
   // the same network as SCL:
   "A6.2" := "A75";
END_REGION

REGION Network 58: Top carriage downward (Top)
   RUNG wire#powerrail
      Contact( "A76" )
      I_Contact( "Alarm" )
      Coil( "A6.3" )
   END_RUNG
   // the same network as SCL:
   "A6.3" := "A76" AND NOT "Alarm";
END_REGION

REGION Network 59: Top carriage brake (Top)
   RUNG wire#powerrail
      Contact( "A85" )
      Coil( "A6.4" )
   END_RUNG
   // the same network as SCL:
   "A6.4" := "A85";
END_REGION

REGION Network 60: Opening clamp to block top film (Top)
   RUNG wire#powerrail
      Contact( "A82" )
      Coil( "A6.5" )
   END_RUNG
   // the same network as SCL:
   "A6.5" := "A82";
END_REGION

REGION Network 61: Closing clamp to block top film (Top)
   RUNG wire#powerrail
      Contact( "A81" )
      Coil( "A6.6" )
   END_RUNG
   // the same network as SCL:
   "A6.6" := "A81";
END_REGION

REGION Network 62: Top cutter forward (Top)
   RUNG wire#powerrail
      Contact( "A79" )
      I_Contact( "Alarm" )
      Coil( "A6.7" )
   END_RUNG
   // the same network as SCL:
   "A6.7" := "A79" AND NOT "Alarm";
END_REGION

REGION Network 63: Top cutter backward (Top)
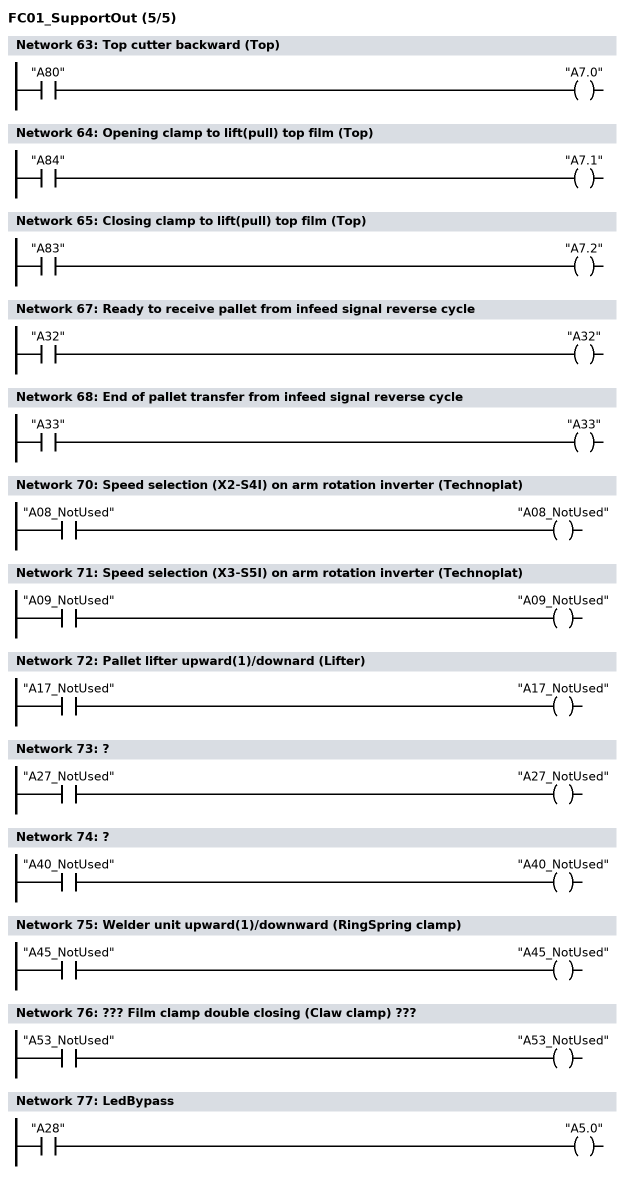
   RUNG wire#powerrail
      Contact( "A80" )
      Coil( "A7.0" )
   END_RUNG
   // the same network as SCL:
   "A7.0" := "A80";
END_REGION

REGION Network 64: Opening clamp to lift(pull) top film (Top)
   RUNG wire#powerrail
      Contact( "A84" )
      Coil( "A7.1" )
   END_RUNG
   // the same network as SCL:
   "A7.1" := "A84";
END_REGION

REGION Network 65: Closing clamp to lift(pull) top film (Top)
   RUNG wire#powerrail
      Contact( "A83" )
      Coil( "A7.2" )
   END_RUNG
   // the same network as SCL:
   "A7.2" := "A83";
END_REGION

REGION Network 66: OTHER
END_REGION

REGION Network 67: Ready to receive pallet from infeed signal reverse cycle
   RUNG wire#powerrail
      Contact( "A32" )
      Coil( "A32" )
   END_RUNG
   // the same network as SCL:
   "A32" := "A32";
END_REGION

REGION Network 68: End of pallet transfer from infeed signal reverse cycle
   RUNG wire#powerrail
      Contact( "A33" )
      Coil( "A33" )
   END_RUNG
   // the same network as SCL:
   "A33" := "A33";
END_REGION

REGION Network 69: OLD (NOT USED)
END_REGION

REGION Network 70: Speed selection (X2-S4I) on arm rotation inverter (Technoplat)
   RUNG wire#powerrail
      Contact( "A08_NotUsed" )
      Coil( "A08_NotUsed" )
   END_RUNG
   // the same network as SCL:
   "A08_NotUsed" := "A08_NotUsed";
END_REGION

REGION Network 71: Speed selection (X3-S5I) on arm rotation inverter (Technoplat)
   RUNG wire#powerrail
      Contact( "A09_NotUsed" )
      Coil( "A09_NotUsed" )
   END_RUNG
   // the same network as SCL:
   "A09_NotUsed" := "A09_NotUsed";
END_REGION

REGION Network 72: Pallet lifter upward(1)/downard (Lifter)
   RUNG wire#powerrail
      Contact( "A17_NotUsed" )
      Coil( "A17_NotUsed" )
   END_RUNG
   // the same network as SCL:
   "A17_NotUsed" := "A17_NotUsed";
END_REGION

REGION Network 73: ?
   RUNG wire#powerrail
      Contact( "A27_NotUsed" )
      Coil( "A27_NotUsed" )
   END_RUNG
   // the same network as SCL:
   "A27_NotUsed" := "A27_NotUsed";
END_REGION

REGION Network 74: ?
   RUNG wire#powerrail
      Contact( "A40_NotUsed" )
      Coil( "A40_NotUsed" )
   END_RUNG
   // the same network as SCL:
   "A40_NotUsed" := "A40_NotUsed";
END_REGION

REGION Network 75: Welder unit upward(1)/downward (RingSpring clamp)
   RUNG wire#powerrail
      Contact( "A45_NotUsed" )
      Coil( "A45_NotUsed" )
   END_RUNG
   // the same network as SCL:
   "A45_NotUsed" := "A45_NotUsed";
END_REGION

REGION Network 76: ??? Film clamp double closing (Claw clamp) ???
   RUNG wire#powerrail
      Contact( "A53_NotUsed" )
      Coil( "A53_NotUsed" )
   END_RUNG
   // the same network as SCL:
   "A53_NotUsed" := "A53_NotUsed";
END_REGION

REGION Network 77: LedBypass
   RUNG wire#powerrail
      Contact( "A28" )
      Coil( "A5.0" )
   END_RUNG
   // the same network as SCL:
   "A5.0" := "A28";
END_REGION
END_FUNCTION

FUNCTION "FC02_Technoplat_TandC" : Void   // FC2, LAD
TITLE = Technoplat timer and counter
{ S7_Optimized_Access := 'FALSE' }
AUTHOR : Robopac
VERSION : 0.0
// stored: AutoNumber false, IsIECCheckEnabled false, SetENOAutomatically false, UDAEnableTagReadback false
   VAR_INPUT
      FASTSPEED : Bool;
   END_VAR
   VAR_TEMP
      TempInt : Int;
      TempDint : DInt;
   END_VAR
   VAR_TEMP   // added for the SCL form of the ladder/FBD networks
      _w1 : Bool;
      _w2 : Bool;
   END_VAR
BEGIN

REGION Network 1: Time to filter inverter alarms
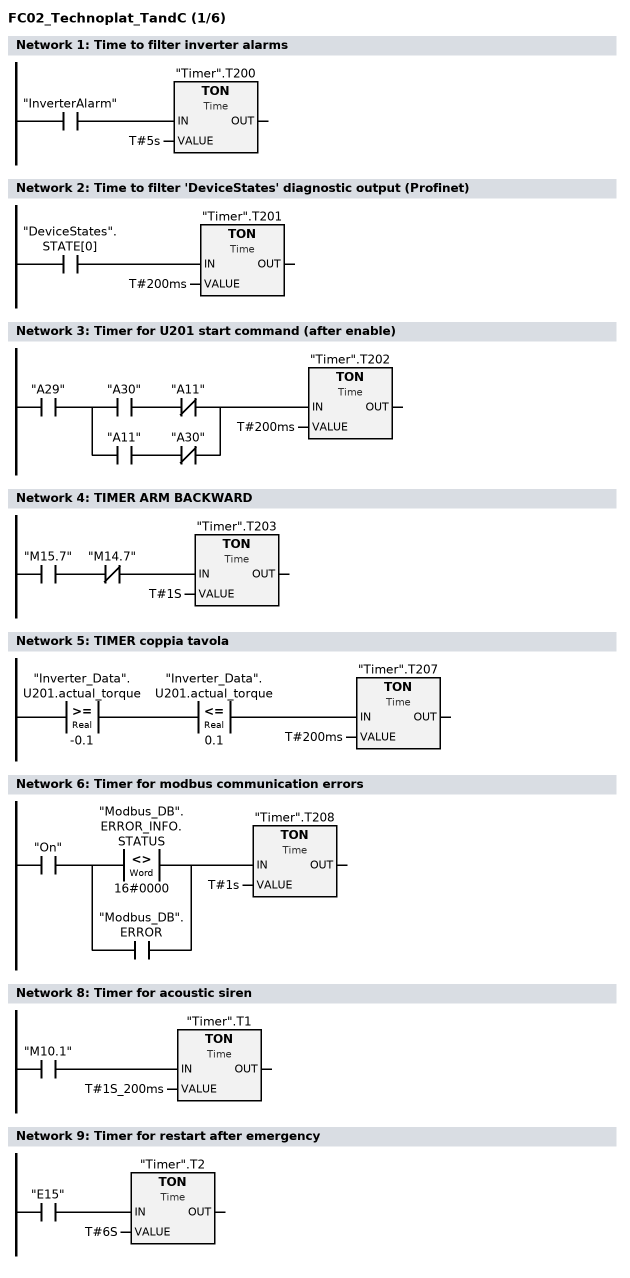
   "Timer".T200.TON(IN := "InverterAlarm", PT := T#5s);   // TON coil
END_REGION

REGION Network 2: Time to filter 'DeviceStates' diagnostic output (Profinet)
   "Timer".T201.TON(IN := "DeviceStates".STATE[0], PT := T#200ms);   // TON coil
END_REGION

REGION Network 3: Timer for U201 start command (after enable)
   "Timer".T202.TON(IN := "A29" AND (("A30" AND NOT "A11") OR ("A11" AND NOT "A30")), PT := T#200ms);   // TON coil
END_REGION

REGION Network 4: TIMER ARM BACKWARD
   "Timer".T203.TON(IN := "M15.7" AND NOT "M14.7", PT := T#1S);   // TON coil
END_REGION

REGION Network 5: TIMER coppia tavola
   "Timer".T207.TON(IN := ("Inverter_Data".U201.actual_torque >= (-0.1)) AND ("Inverter_Data".U201.actual_torque <= 0.1), PT := T#200ms);   // TON coil
END_REGION

REGION Network 6: Timer for modbus communication errors
   "Timer".T208.TON(IN := "On" AND (("Modbus_DB".ERROR_INFO.STATUS <> 16#0000) OR "Modbus_DB".ERROR), PT := T#1s);   // TON coil
END_REGION

REGION Network 7: TECHNOPLAT3000
END_REGION

REGION Network 8: Timer for acoustic siren
   "Timer".T1.TON(IN := "M10.1", PT := T#1S_200ms);   // TON coil
END_REGION

REGION Network 9: Timer for restart after emergency
   "Timer".T2.TON(IN := "E15", PT := T#6S);   // TON coil
END_REGION

REGION Network 10: Timer to reset emergency
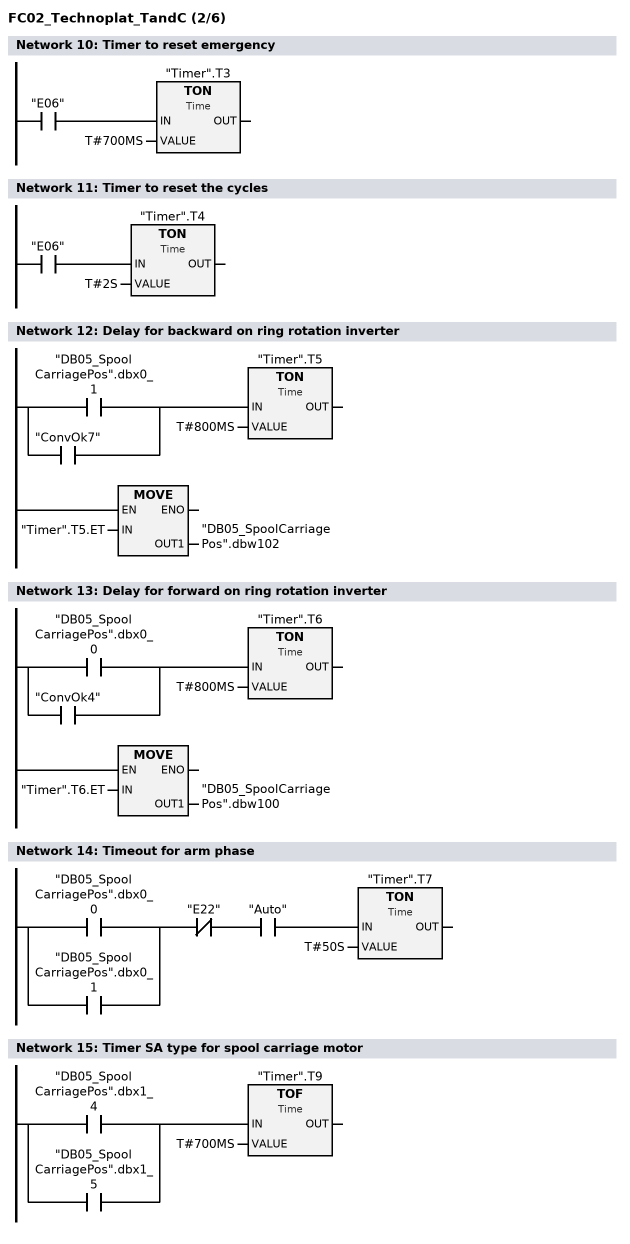
   "Timer".T3.TON(IN := "E06", PT := T#700MS);   // TON coil
END_REGION

REGION Network 11: Timer to reset the cycles
   "Timer".T4.TON(IN := "E06", PT := T#2S);   // TON coil
END_REGION

REGION Network 12: Delay for backward on ring rotation inverter
   "Timer".T5.TON(IN := "DB05_SpoolCarriagePos".dbx0_1 OR "ConvOk7", PT := T#800MS);   // TON coil
   "DB05_SpoolCarriagePos".dbw102 := "Timer".T5.ET;
END_REGION

REGION Network 13: Delay for forward on ring rotation inverter
   "Timer".T6.TON(IN := "DB05_SpoolCarriagePos".dbx0_0 OR "ConvOk4", PT := T#800MS);   // TON coil
   "DB05_SpoolCarriagePos".dbw100 := "Timer".T6.ET;
END_REGION

REGION Network 14: Timeout for arm phase
   "Timer".T7.TON(IN := ("DB05_SpoolCarriagePos".dbx0_0 OR "DB05_SpoolCarriagePos".dbx0_1) AND NOT "E22" AND "Auto", PT := T#50S);   // TON coil
END_REGION

REGION Network 15: Timer SA type for spool carriage motor
   "Timer".T9.TOF(IN := "DB05_SpoolCarriagePos".dbx1_4 OR "DB05_SpoolCarriagePos".dbx1_5, PT := T#700MS);   // TOF coil
END_REGION

REGION Network 16: Timer SA type for arm rotation motor
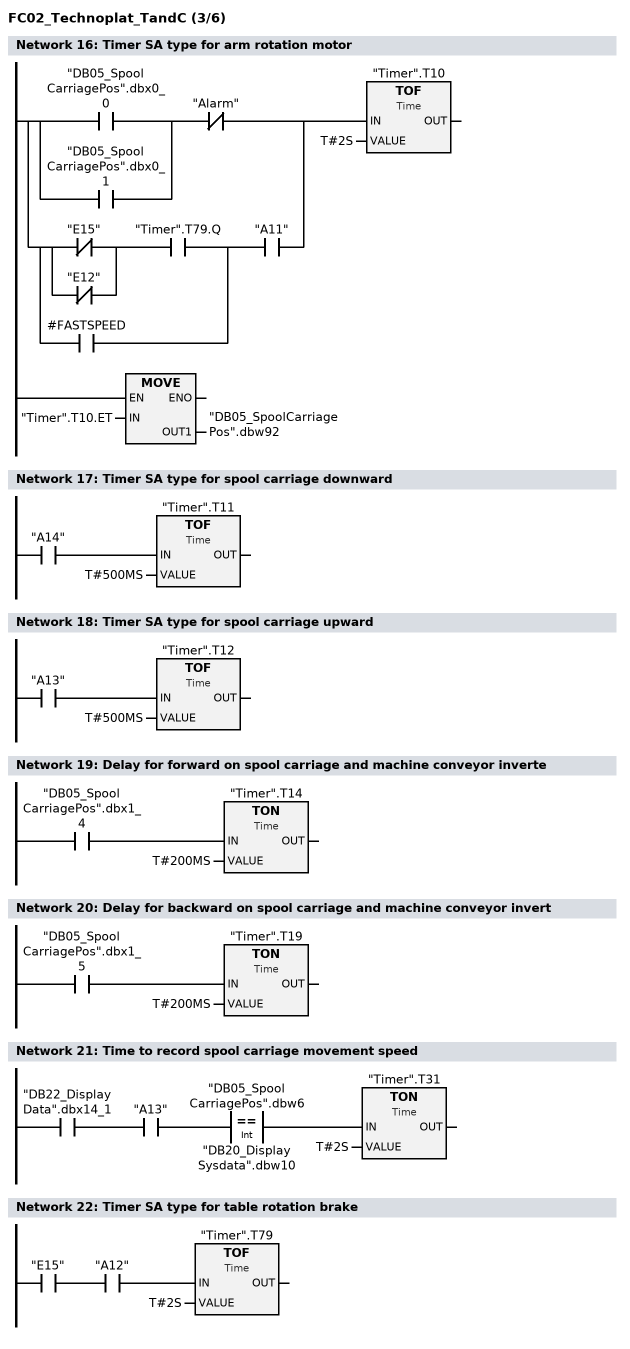
   "Timer".T10.TOF(IN := (("DB05_SpoolCarriagePos".dbx0_0 OR "DB05_SpoolCarriagePos".dbx0_1) AND NOT "Alarm") OR ((((NOT "E15" OR NOT "E12") AND "Timer".T79.Q) OR #FASTSPEED) AND "A11"), PT := T#2S);   // TOF coil
   "DB05_SpoolCarriagePos".dbw92 := "Timer".T10.ET;
END_REGION

REGION Network 17: Timer SA type for spool carriage downward
   "Timer".T11.TOF(IN := "A14", PT := T#500MS);   // TOF coil
END_REGION

REGION Network 18: Timer SA type for spool carriage upward
   "Timer".T12.TOF(IN := "A13", PT := T#500MS);   // TOF coil
END_REGION

REGION Network 19: Delay for forward on spool carriage and machine conveyor inverte
   "Timer".T14.TON(IN := "DB05_SpoolCarriagePos".dbx1_4, PT := T#200MS);   // TON coil
END_REGION

REGION Network 20: Delay for backward on spool carriage and machine conveyor invert
   "Timer".T19.TON(IN := "DB05_SpoolCarriagePos".dbx1_5, PT := T#200MS);   // TON coil
END_REGION

REGION Network 21: Time to record spool carriage movement speed
   "Timer".T31.TON(IN := "DB22_DisplayData".dbx14_1 AND "A13" AND ("DB05_SpoolCarriagePos".dbw6 = "DB20_DisplaySysdata".dbw10), PT := T#2S);   // TON coil
END_REGION

REGION Network 22: Timer SA type for table rotation brake
   "Timer".T79.TOF(IN := "E15" AND "A12", PT := T#2S);   // TOF coil
END_REGION

REGION Network 23: T87: Timer for slow conveyor manual movement
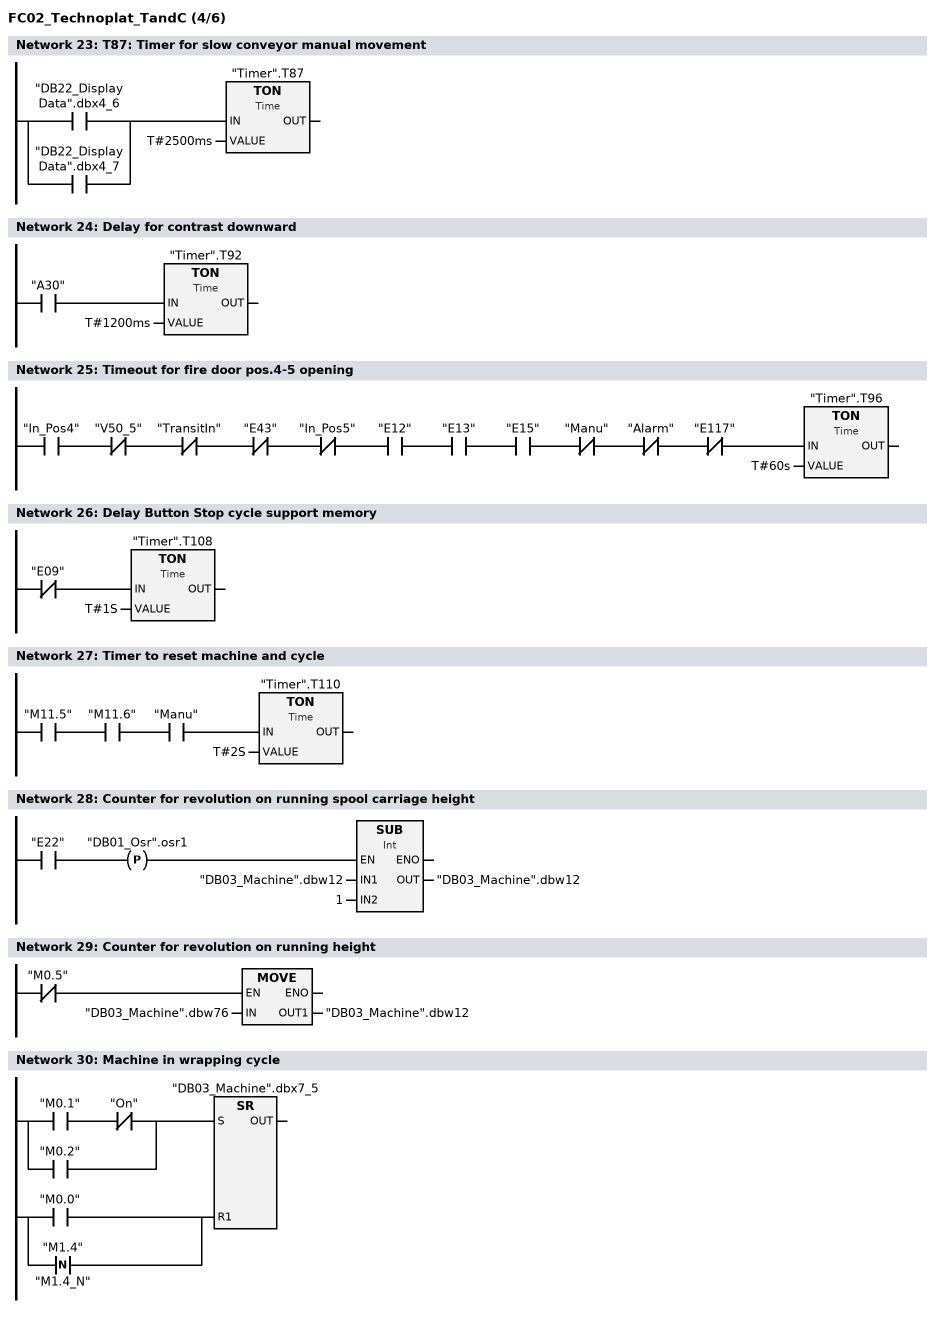
   "Timer".T87.TON(IN := "DB22_DisplayData".dbx4_6 OR "DB22_DisplayData".dbx4_7, PT := T#2500ms);   // TON coil
END_REGION

REGION Network 24: Delay for contrast downward
   "Timer".T92.TON(IN := "A30", PT := T#1200ms);   // TON coil
END_REGION

REGION Network 25: Timeout for fire door pos.4-5 opening
   "Timer".T96.TON(IN := "In_Pos4" AND NOT "V50_5" AND NOT "TransitIn" AND NOT "E43" AND NOT "In_Pos5" AND "E12" AND "E13" AND "E15" AND NOT "Manu" AND NOT "Alarm" AND NOT "E117", PT := T#60s);   // TON coil
END_REGION

REGION Network 26: Delay Button Stop cycle support memory
   "Timer".T108.TON(IN := NOT "E09", PT := T#1S);   // TON coil
END_REGION

REGION Network 27: Timer to reset machine and cycle
   "Timer".T110.TON(IN := "M11.5" AND "M11.6" AND "Manu", PT := T#2S);   // TON coil
END_REGION

REGION Network 28: Counter for revolution on running spool carriage height
   RUNG wire#powerrail
      Contact( "E22" )
      P_Trig( "DB01_Osr".osr1 )
      { S7_Templates := "SrcType := Int"; S7_GenerateENO := "TRUE" } Sub(in1 := "DB03_Machine".dbw12, in2 := 1, out => "DB03_Machine".dbw12)
   END_RUNG
   // the same network as SCL:
   #_w1 := "E22" AND NOT "DB01_Osr".osr1;   // rising edge
   "DB01_Osr".osr1 := "E22";
   IF #_w1 THEN "DB03_Machine".dbw12 := "DB03_Machine".dbw12 - 1; END_IF;
END_REGION

REGION Network 29: Counter for revolution on running height
   RUNG wire#powerrail
      I_Contact( "M0.5" )
      { S7_GenerateENO := "TRUE" } Move(in := "DB03_Machine".dbw76, out1 => "DB03_Machine".dbw12)
   END_RUNG
   // the same network as SCL:
   IF NOT "M0.5" THEN "DB03_Machine".dbw12 := "DB03_Machine".dbw76; END_IF;
END_REGION

REGION Network 30: Machine in wrapping cycle
   RUNG wire#powerrail
      Contact( "M0.1" )
      I_Contact( "On" )
      wire#w1
      S_SR(operand := "DB03_Machine".dbx7_5, r1 := wire#w2)
   END_RUNG
   RUNG wire#powerrail
      Contact( "M0.2" )
   END_RUNG wire#w1
   RUNG wire#powerrail
      Contact( "M0.0" )
   END_RUNG wire#w2
   RUNG wire#powerrail
      N_Contact(operand := "M1.4", bit := "M1.4_N")
   END_RUNG wire#w2
   // the same network as SCL:
   #_w1 := NOT "M1.4" AND "M1.4_N";   // falling edge of "M1.4"
   "M1.4_N" := "M1.4";
   IF ("M0.1" AND NOT "On") OR "M0.2" THEN
       "DB03_Machine".dbx7_5 := TRUE;   // SR flip-flop
   END_IF;
   IF "M0.0" OR #_w1 THEN "DB03_Machine".dbx7_5 := FALSE; END_IF;
END_REGION

REGION Network 31: Support memory to refresh pallet per hour value
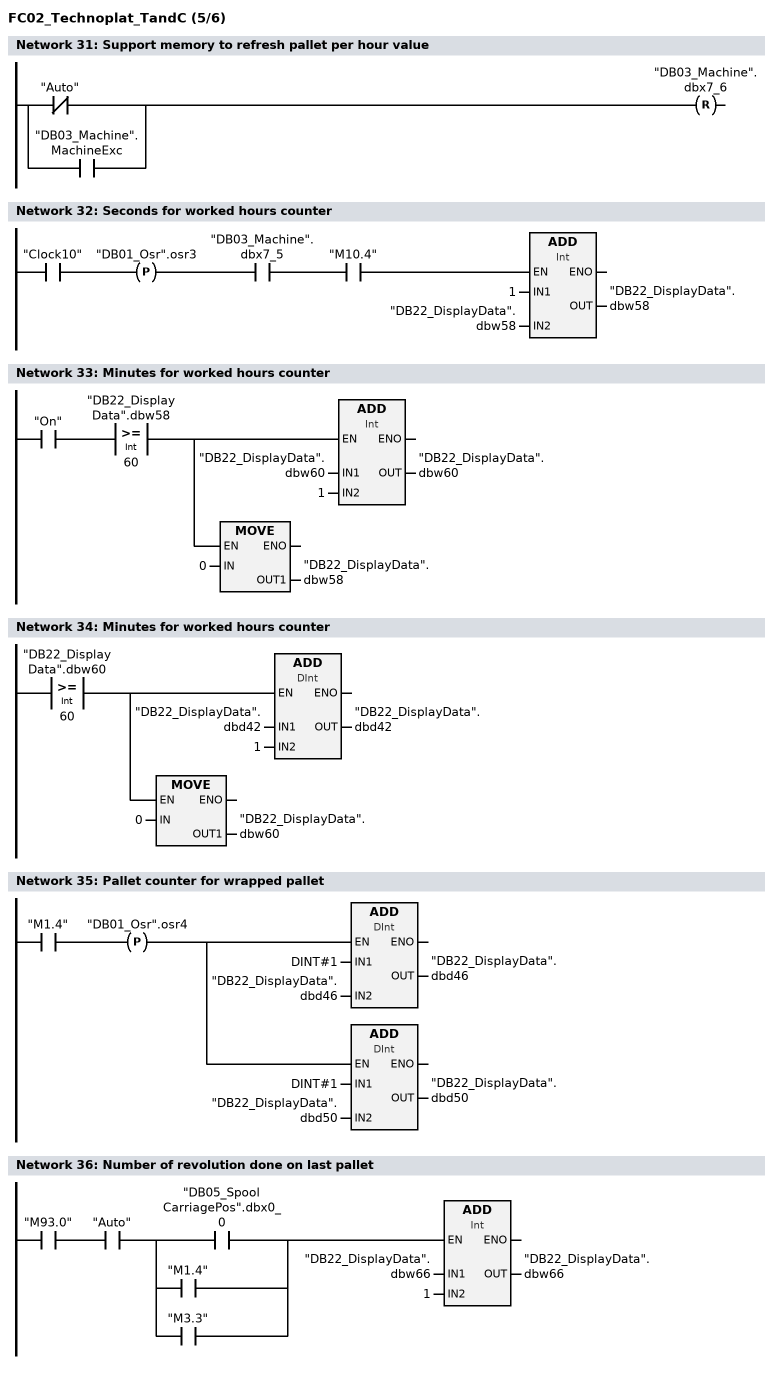
   RUNG wire#powerrail
      I_Contact( "Auto" )
      wire#w1
      R_Coil( "DB03_Machine".dbx7_6 )
   END_RUNG
   RUNG wire#powerrail
      Contact( "DB03_Machine".MachineExc )
   END_RUNG wire#w1
   // the same network as SCL:
   IF NOT "Auto" OR "DB03_Machine".MachineExc THEN "DB03_Machine".dbx7_6 := FALSE; END_IF;
END_REGION

REGION Network 32: Seconds for worked hours counter
   RUNG wire#powerrail
      Contact( "Clock10" )
      P_Trig( "DB01_Osr".osr3 )
      Contact( "DB03_Machine".dbx7_5 )
      Contact( "M10.4" )
      { S7_Templates := "SrcType := Int"; S7_GenerateENO := "TRUE" } Add(in1 := 1, in2 := "DB22_DisplayData".dbw58, out => "DB22_DisplayData".dbw58)
   END_RUNG
   // the same network as SCL:
   #_w1 := "Clock10" AND NOT "DB01_Osr".osr3;   // rising edge
   "DB01_Osr".osr3 := "Clock10";
   IF #_w1 AND "DB03_Machine".dbx7_5 AND "M10.4" THEN
       "DB22_DisplayData".dbw58 := 1 + "DB22_DisplayData".dbw58;
   END_IF;
END_REGION

REGION Network 33: Minutes for worked hours counter
   RUNG wire#powerrail
      Contact( "On" )
      { S7_Templates := "SrcType := Int" } GE_Contact(in1 := "DB22_DisplayData".dbw58, in2 := 60)
      wire#w1
      { S7_Templates := "SrcType := Int"; S7_GenerateENO := "TRUE" } Add(in1 := "DB22_DisplayData".dbw60, in2 := 1, out => "DB22_DisplayData".dbw60)
   END_RUNG
   RUNG wire#w1
      { S7_GenerateENO := "TRUE" } Move(in := 0, out1 => "DB22_DisplayData".dbw58)
   END_RUNG
   // the same network as SCL:
   IF "On" AND ("DB22_DisplayData".dbw58 >= 60) THEN
       "DB22_DisplayData".dbw60 := "DB22_DisplayData".dbw60 + 1;
       "DB22_DisplayData".dbw58 := 0;
   END_IF;
END_REGION

REGION Network 34: Minutes for worked hours counter
   RUNG wire#powerrail
      { S7_Templates := "SrcType := Int" } GE_Contact(in1 := "DB22_DisplayData".dbw60, in2 := 60)
      wire#w1
      { S7_Templates := "SrcType := DInt"; S7_GenerateENO := "TRUE" } Add(in1 := "DB22_DisplayData".dbd42, in2 := 1, out => "DB22_DisplayData".dbd42)
   END_RUNG
   RUNG wire#w1
      { S7_GenerateENO := "TRUE" } Move(in := 0, out1 => "DB22_DisplayData".dbw60)
   END_RUNG
   // the same network as SCL:
   IF "DB22_DisplayData".dbw60 >= 60 THEN
       "DB22_DisplayData".dbd42 := "DB22_DisplayData".dbd42 + 1;
       "DB22_DisplayData".dbw60 := 0;
   END_IF;
END_REGION

REGION Network 35: Pallet counter for wrapped pallet
   RUNG wire#powerrail
      Contact( "M1.4" )
      P_Trig( "DB01_Osr".osr4 )
      wire#w1
      { S7_Templates := "SrcType := DInt"; S7_GenerateENO := "TRUE" } Add(in1 := DINT#1, in2 := "DB22_DisplayData".dbd46, out => "DB22_DisplayData".dbd46)
   END_RUNG
   RUNG wire#w1
      { S7_Templates := "SrcType := DInt"; S7_GenerateENO := "TRUE" } Add(in1 := DINT#1, in2 := "DB22_DisplayData".dbd50, out => "DB22_DisplayData".dbd50)
   END_RUNG
   // the same network as SCL:
   #_w1 := "M1.4" AND NOT "DB01_Osr".osr4;   // rising edge
   "DB01_Osr".osr4 := "M1.4";
   IF #_w1 THEN
       "DB22_DisplayData".dbd46 := DINT#1 + "DB22_DisplayData".dbd46;
       "DB22_DisplayData".dbd50 := DINT#1 + "DB22_DisplayData".dbd50;
   END_IF;
END_REGION

REGION Network 36: Number of revolution done on last pallet
   RUNG wire#powerrail
      Contact( "M93.0" )
      Contact( "Auto" )
      wire#w1
      Contact( "DB05_SpoolCarriagePos".dbx0_0 )
      wire#w2
      { S7_Templates := "SrcType := Int"; S7_GenerateENO := "TRUE" } Add(in1 := "DB22_DisplayData".dbw66, in2 := 1, out => "DB22_DisplayData".dbw66)
   END_RUNG
   RUNG wire#w1
      Contact( "M1.4" )
   END_RUNG wire#w2
   RUNG wire#w1
      Contact( "M3.3" )
   END_RUNG wire#w2
   // the same network as SCL:
   IF "M93.0" AND "Auto" AND ("DB05_SpoolCarriagePos".dbx0_0 OR "M1.4" OR "M3.3") THEN
       "DB22_DisplayData".dbw66 := "DB22_DisplayData".dbw66 + 1;
   END_IF;
END_REGION

REGION Network 37: Number of revolution done on last pallet
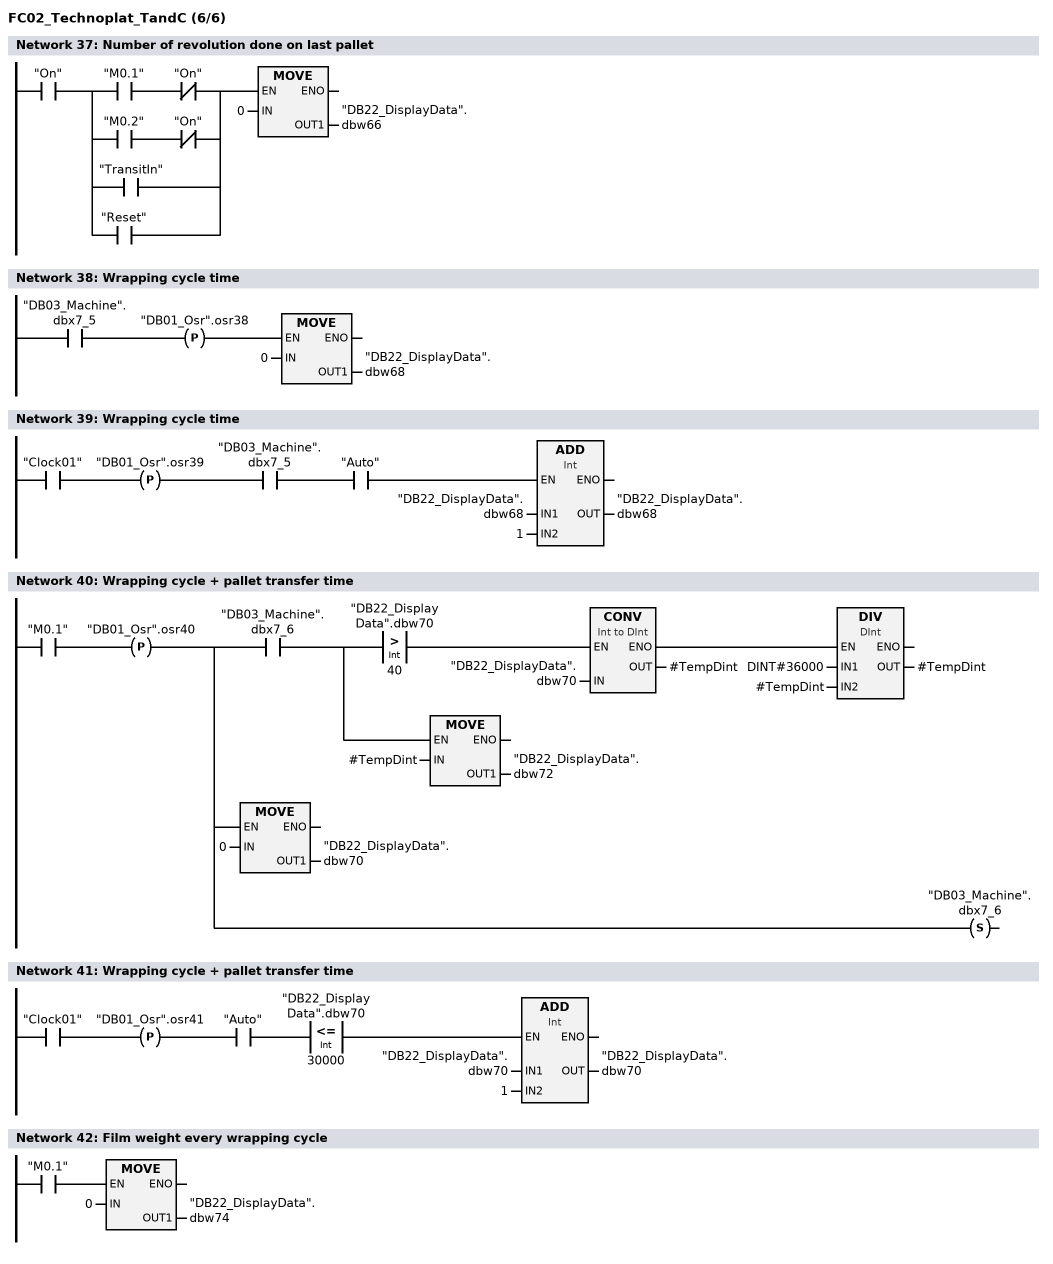
   RUNG wire#powerrail
      Contact( "On" )
      wire#w1
      Contact( "M0.1" )
      I_Contact( "On" )
      wire#w2
      { S7_GenerateENO := "TRUE" } Move(in := 0, out1 => "DB22_DisplayData".dbw66)
   END_RUNG
   RUNG wire#w1
      Contact( "M0.2" )
      I_Contact( "On" )
   END_RUNG wire#w2
   RUNG wire#w1
      Contact( "TransitIn" )
   END_RUNG wire#w2
   RUNG wire#w1
      Contact( "Reset" )
   END_RUNG wire#w2
   // the same network as SCL:
   IF "On" AND (("M0.1" AND NOT "On") OR ("M0.2" AND NOT "On") OR "TransitIn" OR "Reset") THEN
       "DB22_DisplayData".dbw66 := 0;
   END_IF;
END_REGION

REGION Network 38: Wrapping cycle time
   RUNG wire#powerrail
      Contact( "DB03_Machine".dbx7_5 )
      P_Trig( "DB01_Osr".osr38 )
      { S7_GenerateENO := "TRUE" } Move(in := 0, out1 => "DB22_DisplayData".dbw68)
   END_RUNG
   // the same network as SCL:
   #_w1 := "DB03_Machine".dbx7_5 AND NOT "DB01_Osr".osr38;   // rising edge
   "DB01_Osr".osr38 := "DB03_Machine".dbx7_5;
   IF #_w1 THEN "DB22_DisplayData".dbw68 := 0; END_IF;
END_REGION

REGION Network 39: Wrapping cycle time
   RUNG wire#powerrail
      Contact( "Clock01" )
      P_Trig( "DB01_Osr".osr39 )
      Contact( "DB03_Machine".dbx7_5 )
      Contact( "Auto" )
      { S7_Templates := "SrcType := Int"; S7_GenerateENO := "TRUE" } Add(in1 := "DB22_DisplayData".dbw68, in2 := 1, out => "DB22_DisplayData".dbw68)
   END_RUNG
   // the same network as SCL:
   #_w1 := "Clock01" AND NOT "DB01_Osr".osr39;   // rising edge
   "DB01_Osr".osr39 := "Clock01";
   IF #_w1 AND "DB03_Machine".dbx7_5 AND "Auto" THEN
       "DB22_DisplayData".dbw68 := "DB22_DisplayData".dbw68 + 1;
   END_IF;
END_REGION

REGION Network 40: Wrapping cycle + pallet transfer time
   RUNG wire#powerrail
      Contact( "M0.1" )
      P_Trig( "DB01_Osr".osr40 )
      wire#w1
      Contact( "DB03_Machine".dbx7_6 )
      wire#w2
      { S7_Templates := "SrcType := Int" } GT_Contact(in1 := "DB22_DisplayData".dbw70, in2 := 40)
      { S7_Templates := "[SrcType := Int, DestType := DInt]"; S7_GenerateENO := "TRUE" } Convert(in := "DB22_DisplayData".dbw70, out => #TempDint)
      { S7_Templates := "SrcType := DInt"; S7_GenerateENO := "TRUE" } Div(in1 := DINT#36000, in2 := #TempDint, out => #TempDint)
   END_RUNG
   RUNG wire#w2
      { S7_GenerateENO := "TRUE" } Move(in := #TempDint, out1 => "DB22_DisplayData".dbw72)
   END_RUNG
   RUNG wire#w1
      { S7_GenerateENO := "TRUE" } Move(in := 0, out1 => "DB22_DisplayData".dbw70)
   END_RUNG
   RUNG wire#w1
      S_Coil( "DB03_Machine".dbx7_6 )
   END_RUNG
   // the same network as SCL:
   // ENO of a box is taken as its EN; it also drops when the box reports an error
   #_w1 := "M0.1" AND NOT "DB01_Osr".osr40;   // rising edge
   "DB01_Osr".osr40 := "M0.1";
   #_w2 := #_w1 AND "DB03_Machine".dbx7_6;
   IF #_w2 AND ("DB22_DisplayData".dbw70 > 40) THEN
       #TempDint := INT_TO_DINT("DB22_DisplayData".dbw70);
       #TempDint := DINT#36000 / #TempDint;
   END_IF;
   IF #_w2 THEN "DB22_DisplayData".dbw72 := #TempDint; END_IF;
   IF #_w1 THEN
       "DB22_DisplayData".dbw70 := 0;
       "DB03_Machine".dbx7_6 := TRUE;
   END_IF;
END_REGION

REGION Network 41: Wrapping cycle + pallet transfer time
   RUNG wire#powerrail
      Contact( "Clock01" )
      P_Trig( "DB01_Osr".osr41 )
      Contact( "Auto" )
      { S7_Templates := "SrcType := Int" } LE_Contact(in1 := "DB22_DisplayData".dbw70, in2 := 30000)
      { S7_Templates := "SrcType := Int"; S7_GenerateENO := "TRUE" } Add(in1 := "DB22_DisplayData".dbw70, in2 := 1, out => "DB22_DisplayData".dbw70)
   END_RUNG
   // the same network as SCL:
   #_w1 := "Clock01" AND NOT "DB01_Osr".osr41;   // rising edge
   "DB01_Osr".osr41 := "Clock01";
   IF #_w1 AND "Auto" AND ("DB22_DisplayData".dbw70 <= 30000) THEN
       "DB22_DisplayData".dbw70 := "DB22_DisplayData".dbw70 + 1;
   END_IF;
END_REGION

REGION Network 42: Film weight every wrapping cycle
   RUNG wire#powerrail
      Contact( "M0.1" )
      { S7_GenerateENO := "TRUE" } Move(in := 0, out1 => "DB22_DisplayData".dbw74)
   END_RUNG
   // the same network as SCL:
   IF "M0.1" THEN "DB22_DisplayData".dbw74 := 0; END_IF;
END_REGION
END_FUNCTION

FUNCTION "FC03_TechnoplatAux" : Void   // FC3, LAD
TITLE = Auxiliary memory for the machine
{ S7_Optimized_Access := 'FALSE' }
AUTHOR : Robopac
VERSION : 0.0
// stored: AutoNumber false, IsIECCheckEnabled false, SetENOAutomatically false, UDAEnableTagReadback false
   VAR_INPUT
      PHASE : Bool;
   END_VAR
   VAR_TEMP
      Pulse_Reset : Bool;   // Pulse to reset encoders
      SuppSpeed : DWord;
      TempInt_min : Int;
      TempInt_max : Int;
      TempDint : DInt;
   END_VAR
   VAR_TEMP   // added for the SCL form of the ladder/FBD networks
      _w1 : Bool;
      _w2 : Bool;
      _w3 : Bool;
      _w4 : Bool;
   END_VAR
BEGIN

REGION Network 1: OSR and OSF for table phases sensor
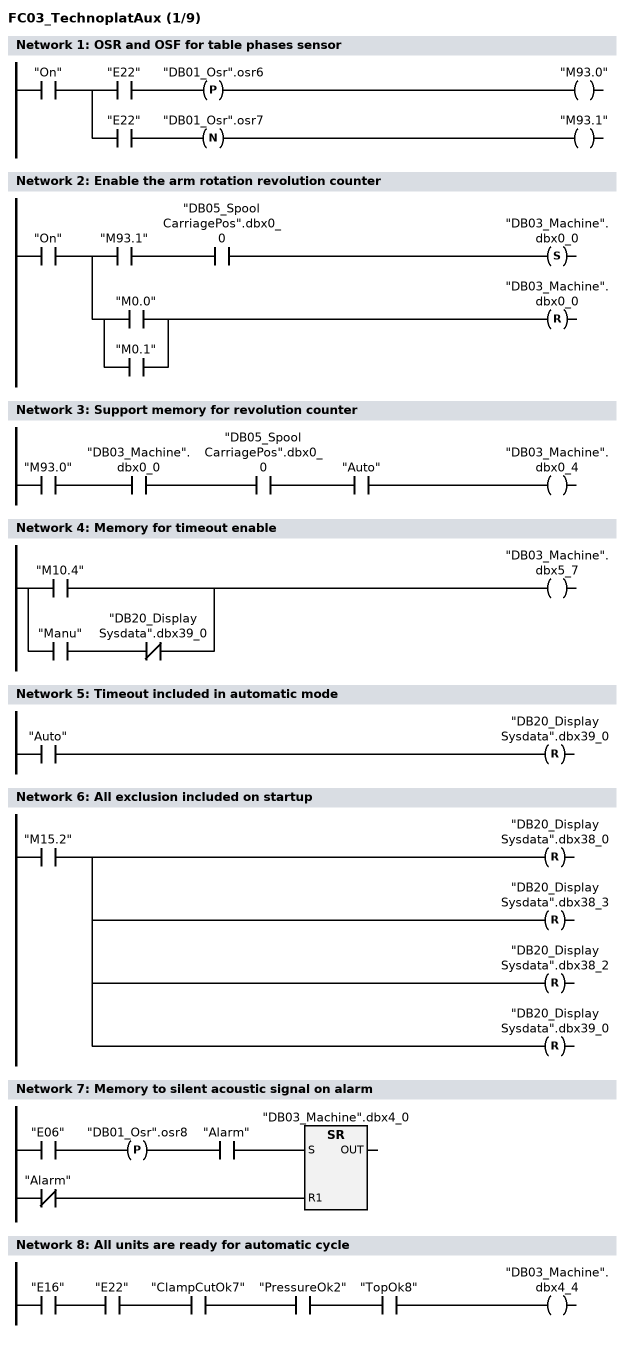
   RUNG wire#powerrail
      Contact( "On" )
      wire#w1
      Contact( "E22" )
      P_Trig( "DB01_Osr".osr6 )
      Coil( "M93.0" )
   END_RUNG
   RUNG wire#w1
      Contact( "E22" )
      N_Trig( "DB01_Osr".osr7 )
      Coil( "M93.1" )
   END_RUNG
   // the same network as SCL:
   #_w1 := "On" AND "E22";
   #_w2 := #_w1 AND NOT "DB01_Osr".osr6;   // rising edge
   "DB01_Osr".osr6 := #_w1;
   "M93.0" := #_w2;
   #_w3 := "On" AND "E22";
   #_w4 := NOT #_w3 AND "DB01_Osr".osr7;   // falling edge
   "DB01_Osr".osr7 := #_w3;
   "M93.1" := #_w4;
END_REGION

REGION Network 2: Enable the arm rotation revolution counter
   RUNG wire#powerrail
      Contact( "On" )
      wire#w1
      Contact( "M93.1" )
      Contact( "DB05_SpoolCarriagePos".dbx0_0 )
      S_Coil( "DB03_Machine".dbx0_0 )
   END_RUNG
   RUNG wire#w1
      Contact( "M0.0" )
      wire#w2
      R_Coil( "DB03_Machine".dbx0_0 )
   END_RUNG
   RUNG wire#w1
      Contact( "M0.1" )
   END_RUNG wire#w2
   // the same network as SCL:
   IF "On" AND "M93.1" AND "DB05_SpoolCarriagePos".dbx0_0 THEN "DB03_Machine".dbx0_0 := TRUE; END_IF;
   IF "On" AND ("M0.0" OR "M0.1") THEN "DB03_Machine".dbx0_0 := FALSE; END_IF;
END_REGION

REGION Network 3: Support memory for revolution counter
   RUNG wire#powerrail
      Contact( "M93.0" )
      Contact( "DB03_Machine".dbx0_0 )
      Contact( "DB05_SpoolCarriagePos".dbx0_0 )
      Contact( "Auto" )
      Coil( "DB03_Machine".dbx0_4 )
   END_RUNG
   // the same network as SCL:
   "DB03_Machine".dbx0_4 := "M93.0" AND "DB03_Machine".dbx0_0 AND "DB05_SpoolCarriagePos".dbx0_0 AND "Auto";
END_REGION

REGION Network 4: Memory for timeout enable
   RUNG wire#powerrail
      Contact( "M10.4" )
      wire#w1
      Coil( "DB03_Machine".dbx5_7 )
   END_RUNG
   RUNG wire#powerrail
      Contact( "Manu" )
      I_Contact( "DB20_DisplaySysdata".dbx39_0 )
   END_RUNG wire#w1
   // the same network as SCL:
   "DB03_Machine".dbx5_7 := "M10.4" OR ("Manu" AND NOT "DB20_DisplaySysdata".dbx39_0);
END_REGION

REGION Network 5: Timeout included in automatic mode
   RUNG wire#powerrail
      Contact( "Auto" )
      R_Coil( "DB20_DisplaySysdata".dbx39_0 )
   END_RUNG
   // the same network as SCL:
   IF "Auto" THEN "DB20_DisplaySysdata".dbx39_0 := FALSE; END_IF;
END_REGION

REGION Network 6: All exclusion included on startup
   RUNG wire#powerrail
      Contact( "M15.2" )
      wire#w1
      R_Coil( "DB20_DisplaySysdata".dbx38_0 )
   END_RUNG
   RUNG wire#w1
      R_Coil( "DB20_DisplaySysdata".dbx38_3 )
   END_RUNG
   RUNG wire#w1
      R_Coil( "DB20_DisplaySysdata".dbx38_2 )
   END_RUNG
   RUNG wire#w1
      R_Coil( "DB20_DisplaySysdata".dbx39_0 )
   END_RUNG
   // the same network as SCL:
   IF "M15.2" THEN
       "DB20_DisplaySysdata".dbx38_0 := FALSE;
       "DB20_DisplaySysdata".dbx38_3 := FALSE;
       "DB20_DisplaySysdata".dbx38_2 := FALSE;
       "DB20_DisplaySysdata".dbx39_0 := FALSE;
   END_IF;
END_REGION

REGION Network 7: Memory to silent acoustic signal on alarm
   RUNG wire#powerrail
      Contact( "E06" )
      P_Trig( "DB01_Osr".osr8 )
      Contact( "Alarm" )
      S_SR(operand := "DB03_Machine".dbx4_0, r1 := wire#w1)
   END_RUNG
   RUNG wire#powerrail
      I_Contact( "Alarm" )
   END_RUNG wire#w1
   // the same network as SCL:
   #_w1 := "E06" AND NOT "DB01_Osr".osr8;   // rising edge
   "DB01_Osr".osr8 := "E06";
   IF #_w1 AND "Alarm" THEN
       "DB03_Machine".dbx4_0 := TRUE;   // SR flip-flop
   END_IF;
   IF NOT "Alarm" THEN "DB03_Machine".dbx4_0 := FALSE; END_IF;
END_REGION

REGION Network 8: All units are ready for automatic cycle
   RUNG wire#powerrail
      Contact( "E16" )
      Contact( "E22" )
      Contact( "ClampCutOk7" )
      Contact( "PressureOk2" )
      Contact( "TopOk8" )
      Coil( "DB03_Machine".dbx4_4 )
   END_RUNG
   // the same network as SCL:
   "DB03_Machine".dbx4_4 := "E16" AND "E22" AND "ClampCutOk7" AND "PressureOk2" AND "TopOk8";
END_REGION

REGION Network 9: Prearrangement automatic cycle
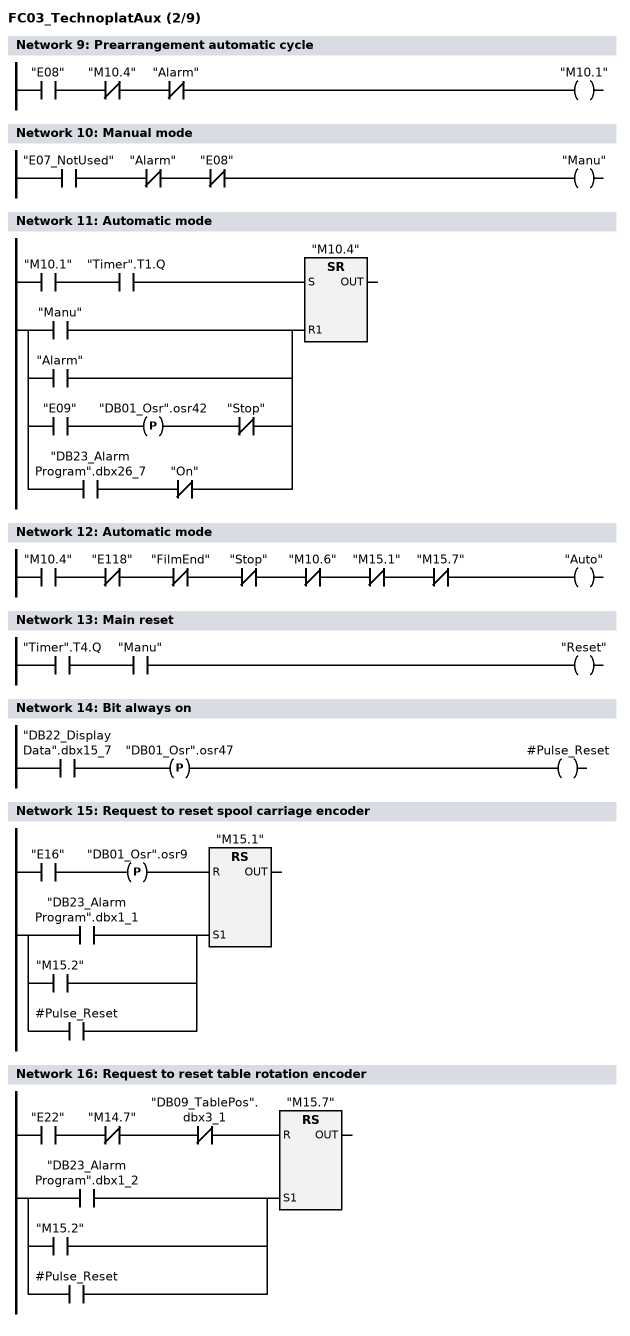
   RUNG wire#powerrail
      Contact( "E08" )
      I_Contact( "M10.4" )
      I_Contact( "Alarm" )
      Coil( "M10.1" )
   END_RUNG
   // the same network as SCL:
   "M10.1" := "E08" AND NOT "M10.4" AND NOT "Alarm";
END_REGION

REGION Network 10: Manual mode
   RUNG wire#powerrail
      Contact( "E07_NotUsed" )
      I_Contact( "Alarm" )
      I_Contact( "E08" )
      Coil( "Manu" )
   END_RUNG
   // the same network as SCL:
   "Manu" := "E07_NotUsed" AND NOT "Alarm" AND NOT "E08";
END_REGION

